//Communication error
	fbKommTof(IN:=bError , PT:=T#20S , Q=> , ET=> );
	fbKommTon(bInput:=fbKommTof.Q , tAlarmDelay:=T#1M , bAutoReset:= , bAlarmOutput=> );
	FAULT :=fbKommTon.bAlarmOutput;
		
//Write busy	
	oaksgvl.aBModbusBusyFlagga[modbusTCP.iModbusLoop,nUnitID] := bBusy;

METHOD mAnalogToRaw : WORD
VAR_INPUT
	rValueToConvert : REAL; //Rå-värde
END_VAR

VAR
	x1 : REAL;
	x2 : REAL;
	y1 : REAL;
	y2 : REAL;
	rPercent : REAL;
	rRawAnalog : REAL;
	rInternalVal: REAL;
END_VAR
//0-100%
rInternalVal := LIMIT(0,rValueToConvert,100);

x1 := 0; 
x2 := 100; 
y1 := 0; 
y2 := 10;
rPercent := fScale2p(rInternalVal,y1, y2, x1, x2);

//0-10V
x1 := 0; 
x2 := 10.24; 
y1 := 0; 
y2 := 32767;
rRawAnalog := fScale2p(rPercent, y1, y2, x1, x2);
mAnalogToRaw := fRealtoWord(rRawAnalog, 1);
END_METHOD

METHOD mAnalogToRawFallback : WORD
VAR_INPUT
	rValueToConvert : REAL; //Rå-värde
END_VAR

VAR
	x1 : REAL;
	x2 : REAL;
	y1 : REAL;
	y2 : REAL;
	rPercent : REAL;
	rRawAnalog : REAL;
	rInternalVal: REAL;
END_VAR
//0-100%
rInternalVal := LIMIT(0,rValueToConvert,100);

//0-10V
x1 := 0; 
x2 := 10.24; 
y1 := 0; 
y2 := 32767;

mAnalogToRawFallback := fRealtoWord(fScale2p(rInternalVal, y1, y2, x1, x2), 1);
END_METHOD

METHOD mRawToAnalog : REAL
VAR_INPUT
	rValueToConvert : WORD; //Rå-värde
END_VAR

VAR
	x1 : REAL;
	x2 : REAL;
	y1 : REAL;
	y2 : REAL;
	rTemp : REAL;
END_VAR
//0-10V
rTemp := fSignedConverter(rValueToConvert);

x1 := 0; 
x2 := 32767;
y1 := 0; 
y2 := 10.24; 
mRawToAnalog := fScale2p(rTemp, y1, y2, x1, x2);
END_METHOD

END_FUNCTION_BLOCK

// oaksModbusLibrary/Metz/fbMetzMR_MULTI
//Oaks AB
//2023-09-19 / Johan Bornemyr
//Funktionsblock för hantering av Metz MR IO-system. 
//MR-MULTI. Modul med 29 IO. Fysisk handställningsmöjlighet 0-10V på modul.
FUNCTION_BLOCK fbMetzMR_MULTI
VAR_INPUT
	bEnable : BOOL := TRUE; //Aktivering
	modbusTCP : ST_ModbusTCP;
	nUnitID: BYTE := 0;
	
	bDO1 : BOOL := FALSE; //Manöver digital utgång 1
	bDO1fallback : BOOL; //Värde vid komm.fel utgång 1
	bDO2 : BOOL := FALSE; //Manöver digital utgång 2
	bDO2fallback : BOOL; //Värde vid komm.fel utgång 2
	bDO3 : BOOL := FALSE; //Manöver digital utgång 3
	bDO3fallback : BOOL; //Värde vid komm.fel utgång 3
	bDO4 : BOOL := FALSE; //Manöver digital utgång 4
	bDO4fallback : BOOL; //Värde vid komm.fel utgång 4
	bTransistorDO1 : BOOL := FALSE; //Manöver digital Transistorutgång 1
	bTransistorDO1fallback : BOOL; //Värde vid komm.fel Transistorutgång 1
	bTransistorDO2 : BOOL := FALSE; //Manöver digital Transistorutgång 2
	bTransistorDO2fallback : BOOL; //Värde vid komm.fel Transistorutgång 2
	bTransistorDO3 : BOOL := FALSE; //Manöver digital Transistorutgång 3
	bTransistorDO3fallback : BOOL; //Värde vid komm.fel Transistorutgång 3
	bTransistorDO4 : BOOL := FALSE; //Manöver digital Transistorutgång 4
	bTransistorDO4fallback : BOOL; //Värde vid komm.fel Transistorutgång 4
	rAO1Setpoint : REAL := 0; //Börvärde Analog utgång 1 (0-100%)
	rAO1FallbackVoltage : REAL := 0; //Börvärde Analog utgång 1 (0-10V)
	rAO2Setpoint : REAL := 0; //Börvärde Analog utgång 2 (0-100%)
	rAO2FallbackVoltage : REAL := 0; //Börvärde Analog utgång 2 (0-10V)
	sensor1config : ST_MetzAI8config;
	sensor2config : ST_MetzAI8config;
	sensor3config : ST_MetzAI8config;
	sensor4config : ST_MetzAI8config;
	sensor5config : ST_MetzAI8config;
	sensor6config : ST_MetzAI8config;
END_VAR
	
VAR_INPUT PERSISTENT
	SP1 AT %M* : REAL := 0;//Komm.fels fördröjning IO~wp:[unit]ms[format]0.0
END_VAR

VAR_OUTPUT
	DI1_V AT %M* : BOOL;//Digital ingång 1~wp:
	DI2_V AT %M* : BOOL;//Digital ingång 2~wp:
	DI3_V AT %M* : BOOL;//Digital ingång 3~wp:
	DI4_V AT %M* : BOOL;//Digital ingång 4~wp:
	DI5_V AT %M* : BOOL;//Digital ingång 5~wp:
	DI6_V AT %M* : BOOL;//Digital ingång 6~wp:
	DI7_V AT %M* : BOOL;//Digital ingång 7~wp:
	DI8_V AT %M* : BOOL;//Digital ingång 8~wp:
	DI9_V AT %M* : BOOL;//Digital ingång 9~wp:
	DI10_V AT %M* : BOOL;//Digital ingång 10~wp:
	DI11_V AT %M* : BOOL;//Digital ingång 11~wp:
	DI12_V AT %M* : BOOL;//Digital ingång 12~wp:
	
	DO1_V AT %M* : BOOL :=FALSE;//Digital utgång 1~wp:
	DO2_V AT %M* : BOOL :=FALSE;//Digital utgång 2~wp:
	DO3_V AT %M* : BOOL :=FALSE;//Digital utgång 3~wp:
	DO4_V AT %M* : BOOL :=FALSE;//Digital utgång 4~wp:
	
	TRANSISTOR_DO1_V AT %M* : BOOL :=FALSE;//Digital utgång 1~wp:
	TRANSISTOR_DO2_V AT %M* : BOOL :=FALSE;//Digital utgång 2~wp:
	TRANSISTOR_DO3_V AT %M* : BOOL :=FALSE;//Digital utgång 3~wp:
	TRANSISTOR_DO4_V AT %M* : BOOL :=FALSE;//Digital utgång 4~wp:
	
	
	AI1_PV AT %M* : REAL; //Råvärde utgång 1~wp:[format]0.00
	AI1_PV1 AT %M* : STRING;//Konfigurering ingång 1~wp:
	sensor1 : ST_MetzAI8Sensor; //Skicka till sensorblock
	AI2_PV AT %M* : REAL; //Råvärde utgång 2~wp:[format]0.00
	AI2_PV1 AT %M* : STRING;//Konfigurering ingång 2~wp:
	sensor2 : ST_MetzAI8Sensor; //Skicka till sensorblock
	AI3_PV AT %M* : REAL; //Råvärde utgång 3~wp:[format]0.00
	AI3_PV1 AT %M* : STRING;//Konfigurering ingång 3~wp:
	sensor3 : ST_MetzAI8Sensor; //Skicka till sensorblock
	AI4_PV AT %M* : REAL; //Råvärde utgång 4~wp:[format]0.00
	AI4_PV1 AT %M* : STRING;//Konfigurering ingång 4~wp:
	sensor4 : ST_MetzAI8Sensor; //Skicka till sensorblock
	AI5_PV AT %M* : REAL; //Råvärde utgång 5~wp:[format]0.00
	AI5_PV1 AT %M* : STRING;//Konfigurering ingång 5~wp:
	sensor5 : ST_MetzAI8Sensor; //Skicka till sensorblock
	AI6_PV AT %M* : REAL; //Råvärde utgång 6~wp:[format]0.00
	AI6_PV1 AT %M* : STRING;//Konfigurering ingång 6~wp:
	sensor6 : ST_MetzAI8Sensor; //Skicka till sensorblock
	
	AO1_OP AT %M* : REAL;//Analog utgång 1~wp:[unit]V[format]0.00
	AO1_FAULT AT %M* : BOOL;//Omkopplare i fel läge utgång 1~wp:
	AO2_OP AT %M* : REAL;//Analog utgång 2~wp:[unit]V[format]0.00
	AO2_FAULT AT %M* : BOOL;//Omkopplare i fel läge utgång 2~wp:
	
	PV8 AT %M* : STRING;//Modbus konfiguering~wp:
	FAULT AT %M* : BOOL;//Kommunikationsfel~wp:
END_VAR
VAR
	//Communication error
	fbKommTof : tof; 
	fbKommTon : fbAlarm;	

	tTimeOut : TIME :=T#5S;
	sIP: STRING(255);
	sPort: STRING(255);
	sModbusID: STRING(255);
	sModbusLoop: STRING(255);
	sTemp : STRING(255);	

	bSekvensFlagga : BOOL;
	R_TRIG_Sekvens: R_TRIG;
(*************** DIGITAL IN - START ***************)	
	FB_MBReadRegs_InputRegsDigitalIn: FB_MBReadInputRegs;
	wInputRegsDigitalIn : WORD; //Read input regs modbus function 4. 	
(*************** DIGITAL IN - SLUT ***************)
(*************** DIGITAL UT - START ***************)
	iStep: INT;
	bError: BOOL;
	bBusy: BOOL;
	
	//Read output values and default values
	FB_MBReadRegs_ArrHolding1: FB_MBReadRegs;
	ArrHolding1 : ARRAY [0..7] OF WORD; //Holding


	fbReadWriteHoldingRegReal_ComError: fbReadWriteHoldingRegReal;
	
	//Configuration
	FB_MBWriteRegs_Config: FB_MBWriteSingleReg;
	wWriteConfig : WORD; //Läs/skriv input regs modbus function 4.
	wReadConfig : WORD; //Läs/skriv input regs modbus function 4.
		
	//Outputs
	FB_MBWriteRegs_Outputs: FB_MBWriteSingleReg;
	wWriteOutputs : WORD; //Läs/skriv input regs modbus function 6.
(*************** DIGITAL UT - SLUT ***************)
(*************** ANALOG UT - START ***************)
	iStepAnalogOut: INT;
	bErrorAnalogOutput: BOOL;
	bBusyAnalogOutput: BOOL;
	
	//Read output values and default values
	FB_MBReadRegs_ArrHoldingAnalogOutput: FB_MBReadRegs;
	ArrHoldingAnalogOutput : ARRAY [0..3] OF WORD; //Holding

	//Outputs in manual mode
	FB_MBReadInputs_wDiscreteInputsAnalogOutput: FB_MBReadInputs;
	wDiscreteInputsAnalogOutput : WORD; //Discrete Input;
	
	fbAlarm_Output1manAnalogOutput : fbAlarm;
	fbAlarm_Output2manAnalogOutput : fbAlarm;

	fbReadWriteHoldingRegReal_ComErrorAnalogOutput: fbReadWriteHoldingRegReal;
	
	//Configuration
	FB_MBWriteRegs_ConfigAnalogOutput: FB_MBWriteRegs;
	wInputRegs2wAnalogOutput : ARRAY[1..2] OF WORD; //Läs/skriv input regs modbus function 16.
	wInputRegs2rAnalogOutput : ARRAY[1..2] OF WORD; //Läs/skriv input regs modbus function 16.
	iConfigChangedAnalogOutput: INT;
	bChangeConfigAnalogOutput: BOOL;
	arrIndexAnalogOutput: INT;
	
	//Outputs
	FB_MBWriteRegs_AnalogOutput: FB_MBWriteRegs;
	wInputRegsOutputswAnalogOutput : ARRAY[1..2] OF WORD; //Läs/skriv input regs modbus function 16.
(*************** ANALOG UT - SLUT ***************)	
(*************** ANALOG IN - START ***************)		
	iStepAnalogIn: INT;
	bErrorAnalogIn: BOOL;
	bBusyAnalogIn: BOOL;	

	//Configuration
	FB_MBReadInputRegs_ValuesAnalogIn: FB_MBReadInputRegs;
	wInputRegsValuesAnalogIn : ARRAY[0..11] OF WORD; //Läs input regs modbus function 4.
	wHoldingRegs2writeConfigAnalogIn : ARRAY[16..21] OF WORD; //Läs/skriv input regs modbus function 16.
	wHoldingRegs2readConfigAnalogIn : ARRAY[16..21] OF WORD; //Läs/skriv input regs modbus function 16.
	
	FB_MBWriteRegs_ConfigAnalogIn: FB_MBWriteRegs;
	FB_MBReadRegs_ConfigAnalogIn: FB_MBReadRegs;
	arrIndexAnalogIn: INT;
	iConfigChangedAnalogIn: INT;
	bChangeConfigAnalogIn: BOOL;

	//Convert to float
	wTempArrayConvertingFromFloatAnalogIn: ARRAY[0..1] OF WORD; // Används för att byta ordning på de två 16-bitars registerna som float-värdet består utav.
(*************** ANALOG IN - SLUT ***************)	
END_VAR

//Sekvens	
	R_TRIG_Sekvens(CLK:= oaksGVL.aBModbusSekvens[modbusTCP.iModbusLoop] = BYTE_TO_INT(nUnitID), Q=> bSekvensFlagga);
	
	
//Modbus config
	sIP := CONCAT (modbusTCP.sIPAddr, '');
	sPort := CONCAT ('<br>Port: ', UINT_TO_STRING(modbusTCP.nTCPPort)); 								
	sModbusID := CONCAT('<br>ID: ', BYTE_TO_STRING(nUnitID));
	sModbusLoop := CONCAT('<br>Loop: ', INT_TO_STRING(modbusTCP.iModbusLoop));	

	sTemp := sIP;
	sTemp := CONCAT(sTemp, sPort);
	sTemp := CONCAT(sTemp, sModbusID);
	sTemp := CONCAT(sTemp, sModbusLoop);
	
	PV8 := sTemp;
	
	mDigitalIn();
	mDigitalOut();
	mAnalogIn();
	mAnalogOut();
	

//Communication error
	fbKommTof(IN:=bErrorAnalogOutput , PT:=T#20S , Q=> , ET=> );
	fbKommTon(bInput:=fbKommTof.Q , tAlarmDelay:=T#1M , bAutoReset:= , bAlarmOutput=> );
	FAULT :=fbKommTon.bAlarmOutput;
		
//Write busy	
	oaksgvl.aBModbusBusyFlagga[modbusTCP.iModbusLoop,nUnitID] := bBusyAnalogOutput;

METHOD PRIVATE config : WORD
VAR_INPUT
	bResistance : BOOL; //0-10V (false) eller resistans (true)
	wSensorType : WORD;
	
END_VAR

VAR
	wOffset : WORD := 0; 
END_VAR
//Temperaturmätning
IF bResistance THEN

	wOffset := wSensorType;
	
	config.0 := FALSE; //Float
	config.1 := wOffset.0; 
	config.2 := wOffset.1; 
	config.3 := wOffset.2; 
	config.4 := wOffset.3;  
	config.5 := wOffset.4; 
	config.6 := wOffset.5; 
	config.7 := TRUE; //Välj resistans 
	config.8 := FALSE; 
	config.9 := FALSE; 
	config.10 := FALSE; 
	config.11 := FALSE; 
	config.12 := FALSE; 
	config.13 := FALSE; 
	config.14 := FALSE; 
	config.15 := FALSE; 
 
  
//Spänningsmätning
ELSE
	config.0 := FALSE; //Float
	config.1 := FALSE; 
	config.2 := FALSE; 
	config.3 := FALSE; 
	config.4 := FALSE;  
	config.5 := FALSE; 
	config.6 := FALSE; 
	config.7 := FALSE; //Välj resistans 
	config.8 := FALSE; 
	config.9 := FALSE; 
	config.10 := FALSE; 
	config.11 := FALSE; 
	config.12 := FALSE; 
	config.13 := FALSE; 
	config.14 := FALSE; 
	config.15 := FALSE; 
END_IF
END_METHOD

METHOD PRIVATE mAnalogIn
VAR_INPUT
END_VAR
	CASE iStepAnalogIn OF

	0: 	//Start/reset
		bBusyAnalogIn := FALSE;
				
		IF bEnable AND bSekvensFlagga THEN
			iStepAnalogIn := 1;
			bErrorAnalogIn := FALSE;
		END_IF
		
	1: 	//Read measured values
		bBusyAnalogIn := TRUE;
			
		FB_MBReadInputRegs_ValuesAnalogIn.bExecute := TRUE;
	
		FB_MBReadInputRegs_ValuesAnalogIn(
		sIPAddr:= modbusTCP.sIpAddr, 
		nTCPPort:= modbusTCP.nTCPPort, 
		nUnitID:= nUnitID, 
		nQuantity:= 12,
		nMBAddr:= 0, 
		cbLength:= SIZEOF(wInputRegsValuesAnalogIn), 
		pDestAddr:= ADR(wInputRegsValuesAnalogIn), 
		bExecute:= , 
		tTimeout:= tTimeOut, 
		bBusy=> , 
		bError=> , 
		nErrId=> , 
		cbRead=> );
		
		//Ingång 1
		wTempArrayConvertingFromFloatAnalogIn[0] := wInputRegsValuesAnalogIn[1];
		wTempArrayConvertingFromFloatAnalogIn[1] := wInputRegsValuesAnalogIn[0]; 

		
		AI1_PV := fWordToReal(wTempArrayConvertingFromFloatAnalogIn);
		
		IF sensor1config.bResistance THEN
			AI1_PV := fWordToReal(wTempArrayConvertingFromFloatAnalogIn);
			AI1_PV1 := CONCAT('Givartyp: ', TO_STRING(sensor1config.sensorType));
		ELSE
			stemp := '0-10V';
			AI1_PV1 := sTemp;
		END_IF
		
		//Info till sensorblock
		sensor1.bComError := FAULT;
		sensor1.rRawValue := AI1_PV;
		sensor1.sSensorConfig := AI1_PV1;
		
		//Ingång 2
		wTempArrayConvertingFromFloatAnalogIn[0] := wInputRegsValuesAnalogIn[3];
		wTempArrayConvertingFromFloatAnalogIn[1] := wInputRegsValuesAnalogIn[2];
		
		AI2_PV := fWordToReal(wTempArrayConvertingFromFloatAnalogIn);
		
		IF sensor2config.bResistance THEN
			AI2_PV1 := CONCAT('Givartyp: ', TO_STRING(sensor2config.sensorType));
		ELSE
			stemp := '0-10V';
			AI2_PV1 := sTemp; 
  
		END_IF
		
		//Info till sensorblock
		sensor2.bComError := FAULT;
		sensor2.rRawValue := AI2_PV;
		sensor2.sSensorConfig := AI2_PV1;
		
		//Ingång 3
		wTempArrayConvertingFromFloatAnalogIn[0] := wInputRegsValuesAnalogIn[5];
		wTempArrayConvertingFromFloatAnalogIn[1] := wInputRegsValuesAnalogIn[4];
		
		AI3_PV := fWordToReal(wTempArrayConvertingFromFloatAnalogIn);
		
		IF sensor3config.bResistance THEN
			AI3_PV1 := CONCAT('Givartyp: ', TO_STRING(sensor3config.sensorType));
		ELSE
			stemp := '0-10V';
			AI3_PV1 := sTemp; 
		END_IF
		
		//Info till sensorblock
		sensor3.bComError := FAULT;
		sensor3.rRawValue := AI3_PV;
		sensor3.sSensorConfig := AI3_PV1;
		
		//Ingång 4
		wTempArrayConvertingFromFloatAnalogIn[0] := wInputRegsValuesAnalogIn[7];
		wTempArrayConvertingFromFloatAnalogIn[1] := wInputRegsValuesAnalogIn[6];
		
		AI4_PV := fWordToReal(wTempArrayConvertingFromFloatAnalogIn);
		
		IF sensor4config.bResistance THEN
			AI4_PV1 := CONCAT('Givartyp: ', TO_STRING(sensor4config.sensorType));
		ELSE
			stemp := '0-10V';
			AI4_PV1 := sTemp;
		END_IF
		
		//Info till sensorblock
		sensor4.bComError := FAULT;
		sensor4.rRawValue := AI4_PV;
		sensor4.sSensorConfig := AI4_PV1;
		
		//Ingång 5
		wTempArrayConvertingFromFloatAnalogIn[0] := wInputRegsValuesAnalogIn[9];
		wTempArrayConvertingFromFloatAnalogIn[1] := wInputRegsValuesAnalogIn[8];

		AI5_PV := fWordToReal(wTempArrayConvertingFromFloatAnalogIn);
	
		IF sensor5config.bResistance THEN
			AI5_PV1 := CONCAT('Givartyp: ', TO_STRING(sensor5config.sensorType));
		ELSE
			stemp := '0-10V';
			AI5_PV1 := sTemp;
		END_IF
		
		//Info till sensorblock
		sensor5.bComError := FAULT;
		sensor5.rRawValue := AI5_PV;
		sensor5.sSensorConfig := AI5_PV1;
		
		//Ingång 6
		wTempArrayConvertingFromFloatAnalogIn[0] := wInputRegsValuesAnalogIn[11];
		wTempArrayConvertingFromFloatAnalogIn[1] := wInputRegsValuesAnalogIn[10]; 
		
		AI6_PV := fWordToReal(wTempArrayConvertingFromFloatAnalogIn);
				
		IF sensor6config.bResistance THEN
			AI6_PV1 := CONCAT('Givartyp: ', TO_STRING(sensor6config.sensorType));
		ELSE
			stemp := '0-10V';
			AI6_PV1 := sTemp;
		END_IF
		
		//Info till sensorblock
		sensor6.bComError := FAULT;
		sensor6.rRawValue := AI6_PV;
		sensor6.sSensorConfig := AI6_PV1;
		
		//Error 
		IF FB_MBReadInputRegs_ValuesAnalogIn.bError THEN
			FB_MBReadInputRegs_ValuesAnalogIn(bExecute := FALSE);
			iStepAnalogIn := 99;
		END_IF
	
		//Gå till nästa steg
		IF NOT FB_MBReadInputRegs_ValuesAnalogIn.bBusy AND NOT FB_MBReadInputRegs_ValuesAnalogIn.bError THEN
			FB_MBReadInputRegs_ValuesAnalogIn(bExecute := FALSE);
			bErrorAnalogIn := FALSE;
			iStepAnalogIn := 2;
		END_IF;
		
	2: 	//Läs config
		bBusyAnalogIn := TRUE;
		FB_MBReadRegs_ConfigAnalogIn.bExecute := TRUE;
	
		//Konfigurering
		wHoldingRegs2writeConfigAnalogIn[16] := config(sensor1config.bResistance,sensor1config.sensorType);
		wHoldingRegs2writeConfigAnalogIn[17] := config(sensor2config.bResistance,sensor2config.sensorType);
		wHoldingRegs2writeConfigAnalogIn[18] := config(sensor3config.bResistance,sensor3config.sensorType);
		wHoldingRegs2writeConfigAnalogIn[19] := config(sensor4config.bResistance,sensor4config.sensorType);
		wHoldingRegs2writeConfigAnalogIn[20] := config(sensor5config.bResistance,sensor5config.sensorType);
		wHoldingRegs2writeConfigAnalogIn[21] := config(sensor6config.bResistance,sensor6config.sensorType);
	
		FB_MBReadRegs_ConfigAnalogIn(
		sIPAddr:= modbusTCP.sIpAddr, 
		nTCPPort:= modbusTCP.nTCPPort, 
		nUnitID:= nUnitID, 
		nQuantity:= 6, 
		nMBAddr:= 16, 
		cbLength:= SIZEOF(wHoldingRegs2readConfigAnalogIn), 
		pDestAddr:= ADR(wHoldingRegs2readConfigAnalogIn), 
		bExecute:= , 
		tTimeout:= tTimeOut, 
		bBusy=> , 
		bError=> , 
		nErrId=> , 
		cbRead=> );

		//Error 
		IF FB_MBReadRegs_ConfigAnalogIn.bError THEN
			FB_MBReadRegs_ConfigAnalogIn(bExecute := FALSE);
			iStepAnalogIn := 99;
		END_IF
	
		//Next step
		IF NOT FB_MBReadRegs_ConfigAnalogIn.bBusy AND NOT FB_MBReadRegs_ConfigAnalogIn.bError THEN
			FB_MBReadRegs_ConfigAnalogIn(bExecute := FALSE);
		
			//Loop to check if config is different
			FOR arrIndexAnalogIn:=16 TO 21 BY 1 DO
				IF wHoldingRegs2readConfigAnalogIn[arrIndexAnalogIn] = wHoldingRegs2writeConfigAnalogIn[arrIndexAnalogIn] THEN
			 		iConfigChangedAnalogIn := iConfigChangedAnalogIn;
				ELSE 
			 		iConfigChangedAnalogIn := iConfigChangedAnalogIn +1;
				END_IF
			END_FOR;
	
			IF iConfigChangedAnalogIn > 0 THEN
				bChangeConfigAnalogIn := TRUE;
				iStepAnalogIn := 3;
				bErrorAnalogIn := FALSE;
			ELSE 
				iStepAnalogIn := 4;
				bErrorAnalogIn := FALSE;
			END_IF
				
		END_IF;
	
	3: //Write if config is different from read value
		bBusyAnalogIn := TRUE;	
		IF bChangeConfigAnalogIn THEN
			FB_MBWriteRegs_ConfigAnalogIn.bExecute := TRUE;
		END_IF
			
		FB_MBWriteRegs_ConfigAnalogIn(
		sIPAddr:= modbusTCP.sIpAddr, 
		nTCPPort:= modbusTCP.nTCPPort, 
		nUnitID:= nUnitID, 
		nQuantity:= 6, 
		nMBAddr:= 16, 
		cbLength:= SIZEOF(wHoldingRegs2writeConfigAnalogIn), 
		pSrcAddr:= ADR(wHoldingRegs2writeConfigAnalogIn), 
		bExecute:=, 
		tTimeout:= tTimeOut, 
		bBusy=> , 
		bError=> , 
		nErrId=> );
		
		IF FB_MBWriteRegs_ConfigAnalogIn.bError THEN
			FB_MBWriteRegs_ConfigAnalogIn(bExecute := FALSE);
			iStepAnalogIn := 99;
		END_IF
	
		//Next step
		IF NOT FB_MBWriteRegs_ConfigAnalogIn.bBusy AND NOT FB_MBWriteRegs_ConfigAnalogIn.bError THEN
			FB_MBWriteRegs_ConfigAnalogIn(bExecute := FALSE);
			iConfigChangedAnalogIn := 0;
			bChangeConfigAnalogIn := FALSE; //Reset write
			bErrorAnalogIn := FALSE;
			iStepAnalogIn := 4;
		END_IF;
			
	4: //Done
		bBusyAnalogIn := FALSE;
		iStepAnalogIn := 0;

	99: //Error handling
		bBusyAnalogIn := FALSE;
		bErrorAnalogIn := TRUE;
		iStepAnalogIn := 0;
		
END_CASE
END_METHOD

METHOD PRIVATE mAnalogOut
VAR_INPUT
END_VAR
	CASE iStepAnalogOut OF

	0: 	//Start/reset
		bBusyAnalogOutput := FALSE;

		IF bEnable AND bSekvensFlagga THEN
			iStepAnalogOut := 1;
			bErrorAnalogOutput := FALSE;
		END_IF
		
	1: 	//Read measured values
		bBusyAnalogOutput := TRUE;
		
		FB_MBReadInputs_wDiscreteInputsAnalogOutput.bExecute := TRUE;

		FB_MBReadInputs_wDiscreteInputsAnalogOutput(
		sIPAddr:= modbusTCP.sIpAddr, 
		nTCPPort:= modbusTCP.nTCPPort, 
		nUnitID:= nUnitID, 
		nQuantity:= 4, 
		nMBAddr:= 0, 
		cbLength:= SIZEOF(wDiscreteInputsAnalogOutput), 
		pDestAddr:= ADR(wDiscreteInputsAnalogOutput),
		bExecute:=, 
		tTimeout:= tTimeOut, 
		bBusy=> , 
		bError=> , 
		nErrId=> , 
		cbRead=> );
	
		//Switch manual alarm
		fbAlarm_Output1manAnalogOutput(bInput:= wDiscreteInputsAnalogOutput.0, tAlarmDelay:= T#3S, bAutoReset:= , bAlarmOutput=> AO1_FAULT);
		fbAlarm_Output2manAnalogOutput(bInput:= wDiscreteInputsAnalogOutput.1, tAlarmDelay:= T#3S, bAutoReset:= , bAlarmOutput=> AO2_FAULT);
			
		//Error 
		IF FB_MBReadInputs_wDiscreteInputsAnalogOutput.bError THEN
			FB_MBReadInputs_wDiscreteInputsAnalogOutput(bExecute := FALSE);
			iStepAnalogOut := 99;
		END_IF
	
		//Next step
		IF NOT FB_MBReadInputs_wDiscreteInputsAnalogOutput.bBusy AND NOT FB_MBReadInputs_wDiscreteInputsAnalogOutput.bError THEN
			FB_MBReadInputs_wDiscreteInputsAnalogOutput(bExecute := FALSE);
			bErrorAnalogOutput := FALSE;
			iStepAnalogOut := 2;
		END_IF;
			
		
	2: //Read Data (Value on output)
		bBusyAnalogOutput := TRUE;
		FB_MBReadRegs_ArrHoldingAnalogOutput.bExecute := TRUE;

		//Read Holding 0-7
		FB_MBReadRegs_ArrHoldingAnalogOutput(
		sIPAddr:= modbusTCP.sIpAddr, 
		nTCPPort:= modbusTCP.nTCPPort, 
		nUnitID:= nUnitID, 
		nQuantity:= 4, 
		nMBAddr:= 74, 
		cbLength:= SIZEOF(ArrHoldingAnalogOutput), 
		pDestAddr:= ADR(ArrHoldingAnalogOutput), 
		bExecute:=, 
		tTimeout:= tTimeOut, 
		bBusy=> ,
		bError=> , 
		nErrId=> , 
		cbRead=> );
	
		//Values
		AO1_OP := mRawToAnalog(ArrHoldingAnalogOutput[0]); //0
		AO2_OP := mRawToAnalog(ArrHoldingAnalogOutput[1]); //1

		//Error 
		IF FB_MBReadRegs_ArrHoldingAnalogOutput.bError THEN
			FB_MBReadRegs_ArrHoldingAnalogOutput(bExecute := FALSE);
			iStepAnalogOut := 99;
		END_IF
	
		//Gå till nästa steg
		IF NOT FB_MBReadRegs_ArrHoldingAnalogOutput.bBusy AND NOT FB_MBReadRegs_ArrHoldingAnalogOutput.bError THEN
			FB_MBReadRegs_ArrHoldingAnalogOutput(bExecute := FALSE);
			bErrorAnalogOutput := FALSE;
			iStepAnalogOut := 3;
		END_IF;

	3: //Read/Write communication error timedelay (config)
		bBusyAnalogOutput := TRUE;

		//User input
		IF SP1 < 0 THEN
			SP1 := 0;
		END_IF;
		
		IF SP1 > 65535 THEN
			SP1 := 655;
		END_IF;
		
		fbReadWriteHoldingRegReal_ComErrorAnalogOutput.bEnable := TRUE;
		
		fbReadWriteHoldingRegReal_ComErrorAnalogOutput(
		sIPAddr:= modbusTCP.sIpAddr, 
		nTCPPort:= modbusTCP.nTCPPort, 
		nUnitID:= nUnitID, 
		mBusAdr:= 66, 
		bEnable:= , 
		tTimeout:= tTimeOut, 
		rReal:= SP1, 
		uiFaktor:= 100, 
		bError=> , 
		bBusy=> , 
		bSuccess=> );
				
		//Error 
		IF fbReadWriteHoldingRegReal_ComErrorAnalogOutput.bError THEN
			fbReadWriteHoldingRegReal_ComErrorAnalogOutput(bEnable := FALSE);
			iStepAnalogOut := 99;
		END_IF
	
		//Gå till nästa steg
		IF NOT fbReadWriteHoldingRegReal_ComErrorAnalogOutput.bBusy AND NOT fbReadWriteHoldingRegReal_ComErrorAnalogOutput.bError THEN
			fbReadWriteHoldingRegReal_ComErrorAnalogOutput(bEnable := FALSE);
			bErrorAnalogOutput := FALSE;
			iStepAnalogOut := 4;
		END_IF;

	4:	//Read/Write default values (config)
		
		//Config in IO
		wInputRegs2rAnalogOutput[1] := ArrHoldingAnalogOutput[2]; //3;
		wInputRegs2rAnalogOutput[2] := ArrHoldingAnalogOutput[3]; //4;
		//Config in PLC	
		wInputRegs2wAnalogOutput[1] := mAnalogToRawFallback(rAO1FallbackVoltage); //3;
		wInputRegs2wAnalogOutput[2] := mAnalogToRawFallback(rAO2FallbackVoltage); //4;
		
		FOR arrIndexAnalogOutput:=1 TO 2 BY 1 DO
				IF wInputRegs2rAnalogOutput[arrIndexAnalogOutput] = wInputRegs2wAnalogOutput[arrIndexAnalogOutput] THEN
			 		iConfigChangedAnalogOutput := iConfigChangedAnalogOutput;
				ELSE 
			 		iConfigChangedAnalogOutput := iConfigChangedAnalogOutput +1;
				END_IF
		END_FOR;
	
		IF iConfigChangedAnalogOutput > 0 THEN
			bChangeConfigAnalogOutput := TRUE;
			iStepAnalogOut := 5;
			bErrorAnalogOutput := FALSE;
		ELSE 
			iStepAnalogOut := 6;
			bErrorAnalogOutput := FALSE;
		END_IF
 
	5: //Write if config is different from read value
		bBusyAnalogOutput := TRUE;	
		IF bChangeConfigAnalogOutput THEN
			FB_MBWriteRegs_ConfigAnalogOutput.bExecute := TRUE;
		END_IF
			
		FB_MBWriteRegs_ConfigAnalogOutput(
		sIPAddr:= modbusTCP.sIpAddr, 
		nTCPPort:= modbusTCP.nTCPPort, 
		nUnitID:= nUnitID, 
		nQuantity:= 2, 
		nMBAddr:= 78, 
		cbLength:= SIZEOF(wInputRegs2wAnalogOutput), 
		pSrcAddr:= ADR(wInputRegs2wAnalogOutput), 
		bExecute:=, 
		tTimeout:= tTimeOut, 
		bBusy=> , 
		bError=> , 
		nErrId=> );
		
		IF FB_MBWriteRegs_ConfigAnalogOutput.bError THEN
			FB_MBWriteRegs_ConfigAnalogOutput(bExecute := FALSE);
			iStepAnalogOut := 99;
		END_IF
	
		//Next step
		IF NOT FB_MBWriteRegs_ConfigAnalogOutput.bBusy AND NOT FB_MBWriteRegs_ConfigAnalogOutput.bError THEN
			FB_MBWriteRegs_ConfigAnalogOutput(bExecute := FALSE);
			iConfigChangedAnalogOutput := 0;
			bChangeConfigAnalogOutput := FALSE; //Reset write
			bErrorAnalogOutput := FALSE;
			iStepAnalogOut := 6;
		END_IF;

	6: //Write outputs
		bBusyAnalogOutput := TRUE;	
			
		wInputRegsOutputswAnalogOutput[1] := mAnalogToRaw(rAO1Setpoint);
		wInputRegsOutputswAnalogOutput[2] := mAnalogToRaw(rAO2Setpoint);
		
		FB_MBWriteRegs_AnalogOutput.bExecute := TRUE;
		
		FB_MBWriteRegs_AnalogOutput(
		sIPAddr:= modbusTCP.sIpAddr, 
		nTCPPort:= modbusTCP.nTCPPort, 
		nUnitID:= nUnitID, 
		nQuantity:= 2, 
		nMBAddr:= 74, 
		cbLength:= SIZEOF(wInputRegsOutputswAnalogOutput), 
		pSrcAddr:= ADR(wInputRegsOutputswAnalogOutput), 
		bExecute:=, 
		tTimeout:= tTimeOut, 
		bBusy=> , 
		bError=> , 
		nErrId=> );
		
		IF FB_MBWriteRegs_AnalogOutput.bError THEN
			FB_MBWriteRegs_AnalogOutput(bExecute := FALSE);
			iStepAnalogOut := 99;
		END_IF
	
		//Next step
		IF NOT FB_MBWriteRegs_AnalogOutput.bBusy AND NOT FB_MBWriteRegs_AnalogOutput.bError THEN
			FB_MBWriteRegs_AnalogOutput(bExecute := FALSE);
			bErrorAnalogOutput := FALSE;
			iStepAnalogOut := 20;
		END_IF;

	20: //Done
		bBusyAnalogOutput := FALSE;
		iStepAnalogOut := 0;

	99: //Error handling
		bBusyAnalogOutput := FALSE;
		bErrorAnalogOutput := TRUE;
		iStepAnalogOut := 0;
		
END_CASE
END_METHOD

METHOD mAnalogToRaw : WORD
VAR_INPUT
	rValueToConvert : REAL; //Rå-värde
END_VAR

VAR
	x1 : REAL;
	x2 : REAL;
	y1 : REAL;
	y2 : REAL;
	rPercent : REAL;
	rRawAnalog : REAL;
	rInternalVal: REAL;
END_VAR
//0-100%
rInternalVal := LIMIT(0,rValueToConvert,100);

x1 := 0; 
x2 := 100; 
y1 := 0; 
y2 := 10;
rPercent := fScale2p(rInternalVal,y1, y2, x1, x2);

//0-10V
x1 := 0; 
x2 := 10.24; 
y1 := 0; 
y2 := 32767;
rRawAnalog := fScale2p(rPercent, y1, y2, x1, x2);
mAnalogToRaw := fRealtoWord(rRawAnalog, 1);
END_METHOD

METHOD mAnalogToRawFallback : WORD
VAR_INPUT
	rValueToConvert : REAL; //Rå-värde
END_VAR

VAR
	x1 : REAL;
	x2 : REAL;
	y1 : REAL;
	y2 : REAL;
	rPercent : REAL;
	rRawAnalog : REAL;
	rInternalVal: REAL;
END_VAR
//0-100%
rInternalVal := LIMIT(0,rValueToConvert,100);

x1 := 0; 
x2 := 100; 
y1 := 0; 
y2 := 10;
rPercent := fScale2p(rInternalVal,y1, y2, x1, x2);

//0-10V
x1 := 0; 
x2 := 10.24; 
y1 := 0; 
y2 := 32767;

mAnalogToRawFallback := fRealtoWord(fScale2p(rPercent, y1, y2, x1, x2), 1);
END_METHOD

METHOD PRIVATE mDigitalIn
VAR_INPUT
END_VAR
	//Read Input states
	FB_MBReadRegs_InputRegsDigitalIn(
	sIPAddr:= modbusTCP.sIpAddr, 
	nTCPPort:= modbusTCP.nTCPPort, 
	nUnitID:= nUnitID, 
	nQuantity:= 1, 
	nMBAddr:= 70, 
	cbLength:= SIZEOF(wInputRegsDigitalIn), 
	pDestAddr:= ADR(wInputRegsDigitalIn), 
	bExecute:= bSekvensFlagga AND bEnable, 
	tTimeout:= tTimeOut, 
	bBusy=> , 
	bError=> , 
	nErrId=> , 
	cbRead=> );
	
	DI1_V := wInputRegsDigitalIn.0;
	DI2_V := wInputRegsDigitalIn.1;
	DI3_V := wInputRegsDigitalIn.2;
	DI4_V := wInputRegsDigitalIn.3;
	DI5_V := wInputRegsDigitalIn.4;
	DI6_V := wInputRegsDigitalIn.5;
	DI7_V := wInputRegsDigitalIn.6;
	DI8_V := wInputRegsDigitalIn.7;
	DI9_V := wInputRegsDigitalIn.8;
	DI10_V := wInputRegsDigitalIn.9;
	DI11_V := wInputRegsDigitalIn.10;
	DI12_V := wInputRegsDigitalIn.11;
END_METHOD

METHOD PRIVATE mDigitalOut
VAR_INPUT
END_VAR
	CASE iStep OF

	0: 	//Start/reset
		bBusy := FALSE;
						
		IF bEnable AND bSekvensFlagga THEN
			iStep := 1;
			bError := FALSE;
		END_IF
		
	1: //Read Data (Value on output)
		bBusy := TRUE;
		FB_MBReadRegs_ArrHolding1.bExecute := TRUE;

		//Read Values
		FB_MBReadRegs_ArrHolding1(
			sIPAddr:= modbusTCP.sIpAddr, 
			nTCPPort:= modbusTCP.nTCPPort, 
			nUnitID:= nUnitID, 
			nQuantity:= 2, 
			nMBAddr:= 71, 
			cbLength:= SIZEOF(ArrHolding1), 
			pDestAddr:= ADR(ArrHolding1), 
			bExecute:=, 
			tTimeout:= tTimeOut, 
			bBusy=> ,
			bError=> , 
			nErrId=> , 
			cbRead=> );
	
		//Values
		DO1_V := ArrHolding1[0].0;
		DO2_V := ArrHolding1[0].1;
		DO3_V := ArrHolding1[0].2;
		DO4_V := ArrHolding1[0].3;
		TRANSISTOR_DO1_V := ArrHolding1[0].4;
		TRANSISTOR_DO2_V := ArrHolding1[0].5;
		TRANSISTOR_DO3_V := ArrHolding1[0].6;
		TRANSISTOR_DO4_V := ArrHolding1[0].7;

		//Error 
		IF FB_MBReadRegs_ArrHolding1.bError THEN
			FB_MBReadRegs_ArrHolding1(bExecute := FALSE);
			iStep := 99;
		END_IF
	
		//Gå till nästa steg
		IF NOT FB_MBReadRegs_ArrHolding1.bBusy AND NOT FB_MBReadRegs_ArrHolding1.bError THEN
			FB_MBReadRegs_ArrHolding1(bExecute := FALSE);
			bError := FALSE;
			iStep := 2;
		END_IF;

	2: //Read/Write communication error timedelay (config)
		bBusy := TRUE;

		//User input
		IF SP1 < 0 THEN
			SP1 := 0;
		END_IF;
		
		IF SP1 > 65535 THEN
			SP1 := 655;
		END_IF;
		
		fbReadWriteHoldingRegReal_ComError.bEnable := TRUE;
		
		fbReadWriteHoldingRegReal_ComError(
			sIPAddr:= modbusTCP.sIpAddr, 
			nTCPPort:= modbusTCP.nTCPPort, 
			nUnitID:= nUnitID, 
			mBusAdr:= 66, 
			bEnable:= , 
			tTimeout:= tTimeOut, 
			rReal:= SP1, 
			uiFaktor:= 100, 
			bError=> , 
			bBusy=> , 
			bSuccess=> );
				
		//Error 
		IF fbReadWriteHoldingRegReal_ComError.bError THEN
			fbReadWriteHoldingRegReal_ComError(bEnable := FALSE);
			iStep := 99;
		END_IF
	
		//Gå till nästa steg
		IF NOT fbReadWriteHoldingRegReal_ComError.bBusy AND NOT fbReadWriteHoldingRegReal_ComError.bError THEN
			fbReadWriteHoldingRegReal_ComError(bEnable := FALSE);
			bError := FALSE;
			iStep := 3;
		END_IF;
	
	3:	//Read/Write default values (config)
		//Config in IO
		wReadConfig.0 := ArrHolding1[1].0;
		wReadConfig.1 := ArrHolding1[1].1;
		wReadConfig.2 := ArrHolding1[1].2;
		wReadConfig.3 := ArrHolding1[1].3;
		wReadConfig.4 := ArrHolding1[1].4;
		wReadConfig.5 := ArrHolding1[1].5;
		wReadConfig.6 := ArrHolding1[1].6;
		wReadConfig.7 := ArrHolding1[1].7;
		//Config in PLC	
		wWriteConfig.0 := bDO1fallback; 
		wWriteConfig.1 := bDO2fallback;
		wWriteConfig.2 := bDO3fallback;
		wWriteConfig.3 := bDO4fallback;
		wWriteConfig.4 := bTransistorDO1fallback; 
		wWriteConfig.5 := bTransistorDO2fallback;
		wWriteConfig.6 := bTransistorDO3fallback;
		wWriteConfig.7 := bTransistorDO4fallback;
		
		bBusy := TRUE;	
		IF wReadConfig <> wWriteConfig THEN
			FB_MBWriteRegs_Config.bExecute := TRUE;
		END_IF
		
		FB_MBWriteRegs_Config(
			sIPAddr:= modbusTCP.sIpAddr, 
			nTCPPort:= modbusTCP.nTCPPort, 
			nUnitID:= nUnitID,
			nMBAddr:= 73,
			nValue:= wWriteConfig, 
			bExecute:= , 
			tTimeout:= tTimeout , 
			bBusy=> , 
			bError=> , 
			nErrId=> );
			
		IF FB_MBWriteRegs_Config.bError THEN
			FB_MBWriteRegs_Config(bExecute := FALSE);
			iStep := 99;
		END_IF
	
		//Next step
		IF NOT FB_MBWriteRegs_Config.bBusy AND NOT FB_MBWriteRegs_Config.bError THEN
			FB_MBWriteRegs_Config(bExecute := FALSE);
			bError := FALSE;
			iStep := 4;
		END_IF;

	4: //Write outputs
		bBusy := TRUE;	
			
		wWriteOutputs.0 := bDO1;
		wWriteOutputs.1 := bDO2;
		wWriteOutputs.2 := bDO3;
		wWriteOutputs.3 := bDO4;
		wWriteOutputs.4 := bTransistorDO1;
		wWriteOutputs.5 := bTransistorDO2;
		wWriteOutputs.6 := bTransistorDO3;
		wWriteOutputs.7 := bTransistorDO4;
		
		FB_MBWriteRegs_Outputs.bExecute := TRUE;
		
		FB_MBWriteRegs_Outputs(
			sIPAddr:= modbusTCP.sIpAddr, 
			nTCPPort:= modbusTCP.nTCPPort, 
			nUnitID:= nUnitID,
			nMBAddr:= 71,
			nValue:= wWriteOutputs, 
			bExecute:= , 
			tTimeout:= tTimeout , 
			bBusy=> , 
			bError=> , 
			nErrId=> );
				
		IF FB_MBWriteRegs_Outputs.bError THEN
			FB_MBWriteRegs_Outputs(bExecute := FALSE);
			iStep := 99;
		END_IF
	
		//Next step
		IF NOT FB_MBWriteRegs_Outputs.bBusy AND NOT FB_MBWriteRegs_Outputs.bError THEN
			FB_MBWriteRegs_Outputs(bExecute := FALSE);
			bError := FALSE;
			iStep := 20;
		END_IF;

	20: //Done
		bBusy := FALSE;
		iStep := 0;
		

	99: //Error handling
		bBusy := FALSE;
		bError := TRUE;
		iStep := 0;
		
END_CASE
END_METHOD

METHOD mRawToAnalog : REAL
VAR_INPUT
	rValueToConvert : WORD; //Rå-värde
END_VAR

VAR
	x1 : REAL;
	x2 : REAL;
	y1 : REAL;
	y2 : REAL;
	rTemp : REAL;
END_VAR
//0-10V
rTemp := fSignedConverter(rValueToConvert);

x1 := 0; 
x2 := 32767;
y1 := 0; 
y2 := 10.24; 
mRawToAnalog := fScale2p(rTemp, y1, y2, x1, x2);
END_METHOD

END_FUNCTION_BLOCK

// oaksModbusLibrary/Mitsubishi/fbMitsubishiATA_ATW
//OAKS AB
//2020-05-12
//Funktionsblock för kommunikation med en styrenhet för FLK från Mitshubishi via RS485 (via TCP/IP Gateway)
//Dubbelriktad modbusskrivning för börvärde
FUNCTION_BLOCK fbMitsubishiATA_ATW
VAR_INPUT
	sIPAddr : STRING := ''; 
	nTCPPort : UINT;
	nUnitID : UINT :=1;
	iModbusLoop : INT :=1; //Modbusslinga
	SP AT %M*  : REAL;//Börvärde~wp:[unit]°C[format]0.0[trendoption]i:300
				
END_VAR
VAR_OUTPUT
	
	V AT %M*  : BOOL;//Driftindikering~wp:[trendoptions]i:14400, t:1
	PV AT %M*  : REAL;//Rumstemperatur~wp:[unit]°C[format]0.0[trendoption]i:300
	PV1 AT %M*  : REAL;//Felkod (8000=Inget fel)~wp:[format]0
	PV6 AT %M*  : REAL;//Fläkthastighet~wp:[format]0
	PV7 AT %M*  : REAL;//Driftläge~wp:[format]0
	PV10 AT %M* : STRING;//Modbus konfiguering~wp:
	AL AT %M* : BOOL;//Summalarm~wp:
	FAULT AT %M* : BOOL;//Kommunikationsfel~wp:
	
END_VAR
VAR
	offset : WORD;
	rTemp : REAL;
	iTemp : UINT;
	bSekvensFlagga : BOOL;
			
	fbReadInputRegs_wInputRegs1: FB_MBReadInputRegs;
	wInputRegs1 : WORD; //Holding
		
	fbReadInputRegs_wInputRegs2: FB_MBReadInputRegs;
	wInputRegs2: WORD;
	
	fbReadRegs_wHolding1: FB_MBReadRegs;
	wArrayHolding1: ARRAY [1..13] OF WORD;
		
	//Kommunikationsfel
	fbKommTof : tof; 
	fbKommTon : ton;
	TON_alarm: TON;

	fbWriteHoldingDoubleControlled_Sp: fbDoubleControlledModbusHolding;
	
	sIP: STRING(255);
	sPort: STRING(255);
	sModbusID: STRING(255);
	sModbusLoop: STRING(255);
	
	sTemp: STRING(255);
END_VAR

//General
	offset := -1;
//Sekvens	
	bSekvensFlagga := oaksGVL.aBModbusSekvens[iModbusLoop] = UINT_TO_INT(nUnitID);
//Modbus konfiguering
	sIP := CONCAT (SIPAddr, '');
	sPort := CONCAT ('<br>Port: ', UINT_TO_STRING(nTCPPort)); 								
	sModbusID := CONCAT('<br>ID: ', UINT_TO_STRING(nUnitID));
	sModbusLoop := CONCAT('<br>Loop: ', INT_TO_STRING(iModbusLoop));

	sTemp := sIP;
	sTemp := CONCAT(sTemp, sPort);
	sTemp := CONCAT(sTemp, sModbusID);
	sTemp := CONCAT(sTemp, sModbusLoop);
		
	PV10 := sTemp;

///////////////		
//READ
///////////////		
	
//Read Inputregs 1
	//Roomtemp
	fbReadInputRegs_wInputRegs1(
	sIPAddr:= sIpAddr, 
	nTCPPort:= INT_TO_UINT(nTCPPort), 
	nUnitID:= INT_TO_BYTE(nUnitID), 
	nQuantity:= 1, 
	nMBAddr:= 1 + offset, 
	cbLength:= SIZEOF(wInputRegs1), 
	pDestAddr:= ADR(wInputRegs1), 
	bExecute:= bSekvensFlagga, 
	tTimeout:= T#3S, 
	bBusy=> , 
	bError=> , 
	nErrId=> , 
	cbRead=> );
	
	//Values
	PV := WORD_TO_REAL(wInputRegs1) / 10;
	
//Read Inputregs 2 
	//Error Code
	fbReadInputRegs_wInputRegs2(
	sIPAddr:= sIpAddr, 
	nTCPPort:= INT_TO_UINT(nTCPPort), 
	nUnitID:= INT_TO_BYTE(nUnitID), 
	nQuantity:= 1, 
	nMBAddr:= 9 + offset, 
	cbLength:= SIZEOF(wInputRegs2), 
	pDestAddr:= ADR(wInputRegs2), 
	bExecute:= bSekvensFlagga, 
	tTimeout:= T#3S, 
	bBusy=> , 
	bError=> , 
	nErrId=> , 
	cbRead=> );
	
	//Values
	PV1 := WORD_TO_REAL(wInputRegs2);
	
	//Error	
	TON_alarm(IN:= (PV1<>8000), PT:= T#1M , Q=> , ET=> );
	AL := TON_alarm.Q;

//Read Holding 1

	//Run
	fbReadRegs_wHolding1(
	sIPAddr:= sIpAddr, 
	nTCPPort:= INT_TO_UINT(nTCPPort), 
	nUnitID:= INT_TO_BYTE(nUnitID), 
	nQuantity:= 13, 
	nMBAddr:= 1 + offset, 
	cbLength:= SIZEOF(wArrayHolding1), 
	pDestAddr:= ADR(wArrayHolding1), 
	bExecute:= bSekvensFlagga, 
	tTimeout:= T#3S, 
	bBusy=> , 
	bError=> , 
	nErrId=> , 
	cbRead=> );
		
	PV6 := wArrayHolding1[1];
	wArrayHolding1[2];
	PV7 := wArrayHolding1[3];
	wArrayHolding1[4];
	wArrayHolding1[5];
	wArrayHolding1[6];
	wArrayHolding1[7];
	V := WORD_TO_BOOL(wArrayHolding1[8]);
	wArrayHolding1[9];
	wArrayHolding1[10];
	wArrayHolding1[11];
	wArrayHolding1[12];
	wArrayHolding1[13];

	
//		
//READ/WRITE Analogue registers		
//

	fbWriteHoldingDoubleControlled_Sp(
	sIPAddr:= sIPAddr, 
	nTCPPort:= nTCPPort, 
	nUnitID:= UINT_TO_BYTE(nUnitID) , 
	nMBAddr:= 2+offset, 
	bExecute:=bSekvensFlagga , 
	rScale:= 10, 
	rWrite:= SP, 
	bBusy=> , 
	bError=> );
	
//Communication error
	fbKommTof(IN:=fbReadInputRegs_wInputRegs1.bError , PT:=T#20S , Q=> , ET=> );
	fbKommTon(IN:=fbKommTof.Q , PT:=T#20M , Q=> , ET=> );
	FAULT :=fbKommTon.Q;
		
//Write busy	
	oaksgvl.aBModbusBusyFlagga[iModbusLoop,nUnitID] := fbReadInputRegs_wInputRegs1.bBusy OR fbReadInputRegs_wInputRegs2.bBusy OR fbWriteHoldingDoubleControlled_Sp.bBusy;

END_FUNCTION_BLOCK

// oaksModbusLibrary/Mitsubishi/fbMitsubishiHydroBox
//OAKS AB
//2020-07-06
//Funktionsblock för kommunikation med en styrenhet HydroBox. 
FUNCTION_BLOCK fbMitsubishiHydroBox
VAR_INPUT
	sIPAddr : STRING := ''; 
	nTCPPort : UINT;
	nUnitID : UINT :=1;
	iModbusLoop : INT :=1; //Modbusslinga
	bStart : BOOL; //Starta värmepump
	bCoolMode : BOOL; //Aktivera kylläge
	rSetpoint : REAL; //Börvärde värme/kyla
				
END_VAR
VAR_OUTPUT
	COMPRESSOR_V AT %M* : BOOL;//Driftindikering~wp:[trendoptions]i:14400, t:1
	COMPRESSOR_OP AT %M* : REAL;//Hastighet~wp:[unit]Hz[format]0[trendoptions]i:300
	PV1 AT %M* : STRING;//Drifläge~wp:[trendoptions]i:14400, t:1	
	SUPPLY_TEMPERATURE_PV AT %M* : REAL;//Utgående vattentemperatur~wp:[unit]°C[format]0.0[trendoptions]i:300
	RETURN_TEMPERATURE_PV AT %M* : REAL;//Ingående vattentemperatur~wp:[unit]°C[format]0.0[trendoptions]i:300
	PV4 AT %M* : REAL;//Utomhusgivare i utedel~wp:[unit]°C[format]0.0[trendoptions]i:300
		
	PV5 AT %M* : REAL;//Larmkod~wp:[format]0[trendoptions]i:300
	PV6 AT %M* : BOOL;//Elpatron 1~wp:[format]0[trendoptions]i:14400, t:1
	PV7 AT %M* : BOOL;//Elpatron 2~wp:[format]0[trendoptions]i:14400, t:1
	
	PV8 AT %M* : STRING;//Modbus konfiguering~wp:
	
	AL AT %M* : BOOL;//Summalarm~wp:
	FAULT AT %M* : BOOL;//Kommunikationsfel~wp:
	
END_VAR
VAR
	itemp2 : INT;
	iTemp : INT;
	rTemp : REAL;
	offset : INT;
	bSekvensFlagga : BOOL;
		
	FB_MBReadRegs_Coils1: FB_MBReadInputs;
	coils1 : BYTE; //Holding	
 
	fbReadInputRegs_wReadRegs1alarm: FB_MBReadRegs;
	wrReadRegs1alarm: WORD;
	TON_alarm: TON;
	
	FB_MBReadRegs_ArrInputRegs1: FB_MBReadInputRegs;
	arrInputRegs1 : ARRAY [0..10] OF WORD; //Input registers
	
	FB_MBReadRegs_ArrHolding1: FB_MBReadRegs;
	ArrHolding1 : ARRAY [0..10] OF WORD; //Holding
	
	fbReadWriteHoldingReg_1: fbReadWriteHoldingReg;
	wWriteHolding1 : WORD;
	
	fbReadWriteHoldingReg_2: fbReadWriteHoldingReg;
	wWriteHolding2 : WORD;
	
	fbReadWriteHoldingReg_3: fbReadWriteHoldingReg;
	wWriteHolding3 : WORD;
	
	//Kommunikationsfel
	fbKommTof : tof; 
	fbKommTon : ton;
	
	//Modbus config
	sIP: STRING(255);
	sPort: STRING(255);
	sModbusID: STRING(255);
	sModbusLoop: STRING(255);
	sTemp : STRING(255);
		
	
	
END_VAR

//General
	offset := -1;
//Sekvens	
	bSekvensFlagga := oaksGVL.aBModbusSekvens[iModbusLoop] = UINT_TO_INT(nUnitID);
//Modbus konfiguering
	sIP := CONCAT (SIPAddr, '');
	sPort := CONCAT ('<br>Port: ', UINT_TO_STRING(nTCPPort)); 								
	sModbusID := CONCAT('<br>ID: ', UINT_TO_STRING(nUnitID));
	sModbusLoop := CONCAT('<br>Loop: ', INT_TO_STRING(iModbusLoop));	

	sTemp := sIP;
	sTemp := CONCAT(sTemp, sPort);
	sTemp := CONCAT(sTemp, sModbusID);
	sTemp := CONCAT(sTemp, sModbusLoop);
	
	PV8 := sTemp;

///////////////		
//READ
///////////////

//COILS

	FB_MBReadRegs_Coils1(
	sIPAddr:= sIpAddr, 
	nTCPPort:= INT_TO_UINT(nTCPPort), 
	nUnitID:= INT_TO_BYTE(nUnitID), 
	nQuantity:= 2, 
	nMBAddr:= 18 + offset, 
	cbLength:= SIZEOF(coils1), 
	pDestAddr:= ADR(coils1), 
	bExecute:= bSekvensFlagga, 
	tTimeout:= T#3S, 
	bBusy=> , 
	bError=> , 
	nErrId=> , 
	cbRead=> );		

		//Values
		PV6 := coils1.0; //0
		PV7 := coils1.1; //1		

//INPUT REGISTERS		
		
//Read Inputregs 1 (Alarm)
	//Error Code
	fbReadInputRegs_wReadRegs1alarm(
	sIPAddr:= sIpAddr, 
	nTCPPort:= INT_TO_UINT(nTCPPort), 
	nUnitID:= INT_TO_BYTE(nUnitID), 
	nQuantity:= 1, 
	nMBAddr:= 13 + offset, 
	cbLength:= SIZEOF(wrReadRegs1alarm), 
	pDestAddr:= ADR(wrReadRegs1alarm), 
	bExecute:= bSekvensFlagga, 
	tTimeout:= T#3S, 
	bBusy=> , 
	bError=> , 
	nErrId=> , 
	cbRead=> );
	
	//Values
	PV5 := WORD_TO_REAL(wrReadRegs1alarm);
	
	//Error	
	TON_alarm(IN:= (PV5<>8000), PT:= T#1M , Q=> , ET=> );
	AL := TON_alarm.Q;		

	//Read input registers 59-63
	FB_MBReadRegs_ArrInputRegs1(
	sIPAddr:= sIpAddr, 
	nTCPPort:= INT_TO_UINT(nTCPPort), 
	nUnitID:= INT_TO_BYTE(nUnitID), 
	nQuantity:= 5, 
	nMBAddr:= 59 + offset, 
	cbLength:= SIZEOF(arrInputRegs1), 
	pDestAddr:= ADR(arrInputRegs1), 
	bExecute:= bSekvensFlagga, 
	tTimeout:= T#3S, 
	bBusy=> , 
	bError=> , 
	nErrId=> , 
	cbRead=> );
		//Values
		rTemp := WORD_TO_REAL(arrInputRegs1[0]); //59
		PV4 := fSignedConverter(rInput:=rTemp ) / 10;
		//arrInputRegs1[1]; //60
		SUPPLY_TEMPERATURE_PV := WORD_TO_REAL(arrInputRegs1[2]) / 100; //61
		//arrInputRegs1[3]; //62
		RETURN_TEMPERATURE_PV := WORD_TO_REAL(arrInputRegs1[4]) / 100; //63
		//arrInputRegs1[5]; //5
		//arrInputRegs1[6]; //6
		//arrInputRegs1[7]; //7
		//arrInputRegs1[8]; //8
		//arrInputRegs1[9]; //9
		//arrInputRegs1[10]; //10

//HOLDING	
	
	//Read Holding 74 (mode)
	FB_MBReadRegs_ArrHolding1(
	sIPAddr:= sIpAddr, 
	nTCPPort:= INT_TO_UINT(nTCPPort), 
	nUnitID:= INT_TO_BYTE(nUnitID), 
	nQuantity:= 1, 
	nMBAddr:= 74 + offset, 
	cbLength:= SIZEOF(ArrHolding1), 
	pDestAddr:= ADR(ArrHolding1), 
	bExecute:= bSekvensFlagga, 
	tTimeout:= T#3S, 
	bBusy=> , 
	bError=> , 
	nErrId=> , 
	cbRead=> );
	
		//Values
		COMPRESSOR_OP := WORD_TO_REAL(ArrHolding1[0]); //0
		COMPRESSOR_V := COMPRESSOR_OP > 0;
		//ArrHolding1[1]; //1
		//ArrHolding1[2]; //2
		//ArrHolding1[3]; //3
		//ArrHolding1[4]; //4
		//ArrHolding1[5]; //5
		//ArrHolding1[6]; //6
		//ArrHolding1[7]; //7
		//ArrHolding1[8]; //8
		//ArrHolding1[9]; //9
		//ArrHolding1[10]; //10

//HOLDING READ/WRITE

	//Read/Write holding (start)
	//0=Av, 1=På
	IF bStart THEN
		wWriteHolding1 := 1;
	ELSE 
		wWriteHolding1 := 0;
	
	END_IF
	
	fbReadWriteHoldingReg_1(
	sIPAddr:= sIpAddr, 
	nTCPPort:= INT_TO_UINT(nTCPPort), 
	nUnitID:= INT_TO_BYTE(nUnitID), 
	mBusAdr:= 26 + offset, 
	bEnable:= bSekvensFlagga, 
	iWrite:= wWriteHolding1, 
	iRead=> , 
	bError=> , 
	bBusy=> );

	//Read/Write holding (heat/cool)
	//1=Värmeläge, 4=kylläge
	IF bCoolMode THEN
		wWriteHolding2 := 4;
		PV1 := 'Kyla';
	ELSE 
		wWriteHolding2 := 1;
		PV1 := 'Värme';
	END_IF
	
	fbReadWriteHoldingReg_2(
	sIPAddr:= sIpAddr, 
	nTCPPort:= INT_TO_UINT(nTCPPort), 
	nUnitID:= INT_TO_BYTE(nUnitID), 
	mBusAdr:= 29 + offset, 
	bEnable:= bSekvensFlagga, 
	iWrite:= wWriteHolding2, 
	iRead=> , 
	bError=> , 
	bBusy=> );
		
	//Read/Write holding (setpoint)
	iTemp := REAL_TO_INT(rSetpoint) * 100;
		
	fbReadWriteHoldingReg_3(
	sIPAddr:= sIpAddr, 
	nTCPPort:= INT_TO_UINT(nTCPPort), 
	nUnitID:= INT_TO_BYTE(nUnitID), 
	mBusAdr:= 33 + offset, 
	bEnable:= bSekvensFlagga, 
	iWrite:= INT_TO_WORD(iTemp), 
	iRead=> , 
	bError=> , 
	bBusy=> );				
	
//Communication error
	fbKommTof(IN:= 	FB_MBReadRegs_Coils1.bError OR
	fbReadInputRegs_wReadRegs1alarm.bError OR
	FB_MBReadRegs_ArrInputRegs1.bError OR
	FB_MBReadRegs_ArrHolding1.bError OR
	fbReadWriteHoldingReg_1.bError OR
	fbReadWriteHoldingReg_2.bError OR
	fbReadWriteHoldingReg_3.bError, 
	PT:=T#20S , Q=> , ET=> );
	fbKommTon(IN:=fbKommTof.Q , PT:=T#20M , Q=> , ET=> );
	FAULT :=fbKommTon.Q;
		
//Write busy	
	oaksgvl.aBModbusBusyFlagga[iModbusLoop,nUnitID] := 
	FB_MBReadRegs_Coils1.bBusy OR
	fbReadInputRegs_wReadRegs1alarm.bBusy OR
	FB_MBReadRegs_ArrInputRegs1.bBusy OR
	FB_MBReadRegs_ArrHolding1.bBusy OR
	fbReadWriteHoldingReg_1.bBusy OR
	fbReadWriteHoldingReg_2.bBusy OR
	fbReadWriteHoldingReg_3.bBusy;

END_FUNCTION_BLOCK

// oaksModbusLibrary/Nicotra Gebhardt/fbNicotraGebhardtRLM
//OAKS AB
//2022-10-31
//Ver. 1.0
//Modbusblock för Nicotra Gebhardt RLM fläkt.
FUNCTION_BLOCK fbNicotraGebhardtRLM
VAR_INPUT
	sIPAddr : STRING := ''; 
	nTCPPort : UINT;
	nUnitID : UINT :=1;
	iModbusLoop : INT :=1; //Modbusslinga
			
END_VAR
VAR_OUTPUT
	RPM AT %M* : REAL;//Varvtal~wp:[unit]RPM[format]0[trendoptions]i:300
	U1 AT %M* : REAL;//Spänning~wp:[unit]V[format]0[trendoptions]i:300
	I1 AT %M* : REAL;//Ampere~wp:[unit]A[format]0.0[trendoptions]i:300	
	P1 AT %M* : REAL;//Effekt~wp:[unit]kW[format]0.0[trendoptions]i:300	
	E1 AT %M* : REAL;//Energi~wp:[unit]kWh[format]0.0[trendoptions]i:300		
	PV8 AT %M* : STRING;//Modbus konfiguering~wp:
	FAULT AT %M* : BOOL;//Kommunikationsfel~wp:[alarmoptions]p:2
	
END_VAR
VAR
	offset : UINT;
	rTemp1 : REAL;	
	rTemp2 : REAL;	
	rTemp3 : REAL;	
	bSekvensFlagga : BOOL;
			
	FB_MBReadRegs_ArrReadInputsRegs1 : FB_MBReadInputRegs;	
	wArrReadInputsRegs1 : ARRAY [0..33] OF WORD; //ReadInputsRegs
		
	//Kommunikationsfel
	fbKommTof : tof; 
	fbKommTon : fbAlarm;
	
	sIP: STRING(255);
	sPort: STRING(255);
	sModbusID: STRING(255);
	sModbusLoop: STRING(255);
	sTemp : STRING(255);
	
END_VAR

//General
	offset := 0;
//Sekvens	
	bSekvensFlagga := oaksGVL.aBModbusSekvens[iModbusLoop] = UINT_TO_INT(nUnitID);
//Modbus konfiguering
	sIP := CONCAT (SIPAddr, '');
	sPort := CONCAT ('<br>Port: ', UINT_TO_STRING(nTCPPort)); 								
	sModbusID := CONCAT('<br>ID: ', UINT_TO_STRING(nUnitID));
	sModbusLoop := CONCAT('<br>Loop: ', INT_TO_STRING(iModbusLoop));	

	sTemp := sIP;
	sTemp := CONCAT(sTemp, sPort);
	sTemp := CONCAT(sTemp, sModbusID);
	sTemp := CONCAT(sTemp, sModbusLoop);
	
	PV8 := sTemp;

///////////////		
//READ
///////////////		
	
	//Read Inputs 0-33
	FB_MBReadRegs_ArrReadInputsRegs1(
	sIPAddr:= sIpAddr, 
	nTCPPort:= (nTCPPort), 
	nUnitID:= UINT_TO_BYTE(nUnitID), 
	nQuantity:= 34, 
	nMBAddr:= 0 + offset,
	cbLength:= SIZEOF(wArrReadInputsRegs1), 
	pDestAddr:= ADR(wArrReadInputsRegs1), 
	bExecute:= bSekvensFlagga,
	tTimeout:= T#10S, 
	bBusy=> , 
	bError=> , 
	nErrId=> , 
	cbRead=> );	
	
		//Values
		//wArrReadInputsRegs1[0]; //0 - Drive Type, Res.:1, Unit:-
		//wArrReadInputsRegs1[1]; //1 - AOC SW version, Res.:0.01, Unit:-
		//wArrReadInputsRegs1[2]; //2 - MOC SW version, Res.:0.01, Unit:-
		//wArrReadInputsRegs1[3]; //3 - PrcOut, Res.:0.01, Unit:%
		RPM := wArrReadInputsRegs1[4]; //4 - RPMOut, (PM) Res.:1, Unit:RPM or (AC)Res.:0.01, Unit:Hz
		//wArrReadInputsRegs1[5]; //5 - Intern Temp, Res.:0.01, Unit:ºC
		//wArrReadInputsRegs1[6]; //6 - V In (RMS), Res.:1, Unit:V
		I1 := (wArrReadInputsRegs1[7]*0.001); //7 - I Out, Res.:0.01, Unit:A
		P1 := wArrReadInputsRegs1[8]*0.001; //8 - Power In (filtered), Res.:0.01, Unit:kW
		//wArrReadInputsRegs1[9]*1000; //9 - I Ripple, Res.:0.01, Unit:A
	
		//wArrReadInputsRegs1[10]; //10 - Operation Minutes, Res.:1, Unit:Min
		//wArrReadInputsRegs1[11]; //11 - Operation Day, Res.:1, Unit:Day
		//wArrReadInputsRegs1[12]; //12 - V Ripple, Res.:1, Unit:V
		//wArrReadInputsRegs1[13]; //13 - Config file variant, 2 ASCII characters
		//wArrReadInputsRegs1[14]; //14 - Config file version, Res.:0.01, Unit:-
		//wArrReadInputsRegs1[15]; //15 - ExternSet, Res.:1, Unit:mV
		//wArrReadInputsRegs1[16]; //16 - Power Supply, Res.:1, Unit:V
		//wArrReadInputsRegs1[17]; //17 - OverVoltageCount, Res.:1, Unit:-
		//wArrReadInputsRegs1[18]; //18 - AOC SW variant, Res.:-, Unit:-
		//wArrReadInputsRegs1[19]; //19 - AOC Boot SW, Res.:0.01, Unit:-

		//wArrReadInputsRegs1[20]; //20 - MOC Boot SW, Res.:0.01, Unit:-
		//wArrReadInputsRegs1[21]; //21 - Motor Cfg. Var, Res.:1, Unit:-
		//wArrReadInputsRegs1[22]; //22 - Motor Cfg. Ver., Res.:0.01, Unit:-
		//wArrReadInputsRegs1[23]; //23 - Fan Cfg. Var., Res.:1, Unit:-
		//wArrReadInputsRegs1[24]; //24 - Fan Cfg. Ver, Res.:0.01, Unit:-
		//wArrReadInputsRegs1[25]; //25 - User Data Var., Res.:1, Unit:-
		//wArrReadInputsRegs1[26]; //26 - User Data Ver, Res.:0.01, Unit:-
		//wArrReadInputsRegs1[27]; //27 - IOM SW version, Res.:0.01, Unit:-
		//wArrReadInputsRegs1[28]; //28 - V DC Bus (Peak).:1, Unit:V
		U1 := wArrReadInputsRegs1[29]; //29 - V Motor (Peak), Res.:1, Unit:V

		//wArrReadInputsRegs1[30]*1000; //0 - Power In (unfilterd), Res.:0.01, Unit:kW
		rTemp1 := WORD_TO_REAL (wArrReadInputsRegs1[31]); //1 - Power Consumpt., Res.:1, Unit:Wh
		rTemp2 := WORD_TO_REAL (wArrReadInputsRegs1[32]); //2 - Power Consumpt., Res.:1, Unit:kWh
		rTemp3 := WORD_TO_REAL (wArrReadInputsRegs1[33]); //3 - Power Consumpt., Res.:1, Unit:MWh
		E1 := (((rTemp3 * 1000000) + (rTemp2 * 1000) + rTemp1)*0.001);
	
//Communication error
	fbKommTof(IN:=FB_MBReadRegs_ArrReadInputsRegs1.bError , PT:=T#60S , Q=> , ET=> );
	fbKommTon(bInput:=fbKommTof.Q , tAlarmDelay:=T#20M , bAutoReset:= , bAlarmOutput=> );
	FAULT :=fbKommTon.bAlarmOutput;
		
//Write busy	
	oaksgvl.aBModbusBusyFlagga[iModbusLoop,nUnitID] := FB_MBReadRegs_ArrReadInputsRegs1.bBusy;

END_FUNCTION_BLOCK

// oaksModbusLibrary/Produal/Givare/fbProdualHdhmCo2
//OAKS AB
//2020-03-17
//Funktionsblock för modbus-TCP, Produal HDK-M Koldioxid/temp-givare

FUNCTION_BLOCK fbProdualHdhmCo2
VAR_INPUT
	sIPAddr : STRING := ''; 
	nTCPPort : UINT;
	nUnitID : UINT;
	iModbusLoop : INT :=1; //Modbusslinga
	
END_VAR
VAR_OUTPUT
	PV AT %M*: REAL; //Temperatur~wp:[unit]°C[format]0.0[trendoptions]i:300
	PV1 AT %M* : REAL; //Koldioxidhalt~wp:[unit]ppm[format]0[trendoptions]i:300
	FAULT AT %M*: BOOL; //Kommunikationsfel~wp:
	PV8 AT %M* : STRING;//Modbus konfiguering~wp:
END_VAR
VAR
	
	sIP: STRING(255);
	sPort: STRING(255);
	sModbusID: STRING(255);
	sModbusLoop: STRING(255);
	sTemp : STRING(255);
	iTemp : UINT;
	fbKommTof : tof; 
	fbKommTon : ton;
	fbTempCo2: FB_MBReadInputRegs;
	wTempCo2 : ARRAY[0..1] OF	WORD; 
	bSekvensFlagga : BOOL;
END_VAR
VAR_INPUT PERSISTENT
	rCalTemp : REAL;
	rCalCo2 : REAL;
END_VAR

//Modbus konfiguering
	sIP := CONCAT (SIPAddr, '');
	sPort := CONCAT ('<br>Port: ', UINT_TO_STRING(nTCPPort)); 								
	sModbusID := CONCAT('<br>ID: ', UINT_TO_STRING(nUnitID));
	sModbusLoop := CONCAT('<br>Loop: ', INT_TO_STRING(iModbusLoop));	

	sTemp := sIP;
	sTemp := CONCAT(sTemp, sPort);
	sTemp := CONCAT(sTemp, sModbusID);
	sTemp := CONCAT(sTemp, sModbusLoop);
	
	PV8 := sTemp;

//Sekvens	
	bSekvensFlagga := oaksGVL.aBModbusSekvens[iModbusLoop] = UINT_TO_INT(nUnitID);
	
	fbTempCo2(
	sIPAddr:= sIpAddr, 
	nTCPPort:= INT_TO_UINT(nTCPPort), 
	nUnitID:= INT_TO_BYTE(nUnitID), 
	nQuantity:=2 , 
	nMBAddr:=0 , 
	cbLength:= SIZEOF(wTempCo2), 
	pDestAddr:= ADR(wTempCo2), 
	bExecute:= bSekvensFlagga, 
	tTimeout:= T#20S, 
	bBusy=> , 
	bError=> , 
	nErrId=> , 
	cbRead=> );
	
	fbKommTof(IN:=fbTempCo2.bError , PT:=T#20S , Q=> , ET=> );
	fbKommTon(IN:=fbKommTof.Q , PT:=T#20M , Q=> , ET=> );
	FAULT :=fbKommTon.Q;
	
	//Temp
	iTemp := WORD_TO_UINT(wTempCo2[1]);
	PV := (UINT_TO_REAL(iTemp) /10) + rCalTemp;
	
	//Co2
	iTemp := WORD_TO_UINT(wTempCo2[0]);
	PV1 := (UINT_TO_REAL(iTemp)) + rCalCo2;
	
	//Write busy	
	oaksgvl.aBModbusBusyFlagga[iModbusLoop,nUnitID] := fbTempCo2.bBusy;

END_FUNCTION_BLOCK

// oaksModbusLibrary/Produal/Givare/fbProdualHdhmPirCo2
//OAKS AB
//2021-11-29
//Funktionsblock för modbus-TCP, Produal HDK-M-PIR Koldioxid/temp-givare med inbyggd närvarogivare

FUNCTION_BLOCK fbProdualHdhmPirCo2
VAR_INPUT
	sIPAddr : STRING := ''; 
	nTCPPort : UINT;
	nUnitID : UINT;
	iModbusLoop : INT :=1; //Modbusslinga
	
END_VAR
VAR_OUTPUT
	V AT %M*: BOOL; //Närvaroindikering (fördröjt till och frånslag)~wp:[trendoptions]i:14400, t:1
	PV4 AT %M*: BOOL; //Närvarogivare~wp:[trendoptions]i:14400, t:1
	PV AT %M*: REAL; //Temperatur~wp:[unit]°C[format]0.0[trendoptions]i:300
	PV1 AT %M* : REAL; //Koldioxidhalt~wp:[unit]ppm[format]0[trendoptions]i:300
	FAULT AT %M*: BOOL; //Kommunikationsfel~wp:
	PV8 AT %M* : STRING;//Modbus konfiguering~wp:
END_VAR
VAR
	sIP: STRING(255);
	sPort: STRING(255);
	sModbusID: STRING(255);
	sModbusLoop: STRING(255);
	sTemp : STRING(255);
	iTemp : UINT;
	fbKommTof : tof; 
	fbKommTon : ton;
	fbTempCo2: FB_MBReadInputRegs;
	wTempCo2 : ARRAY[0..1] OF	WORD; 
	bSekvensFlagga : BOOL;
	
	uiStartDelay : UINT;
	uiStopDelay : UINT;
	
	fbWriteStartDelay : fbReadWriteHoldingReg;
	fbWriteStopDelay : fbReadWriteHoldingReg;
	
	fbReadPir : FB_MBReadInputs;
	
	bReadPir : BYTE; // 10002 PIR sensor state (immediate) - 10003 PIR sensor state (control)
END_VAR
VAR_INPUT PERSISTENT
	rCalTemp : REAL;
	rCalCo2 : REAL;
END_VAR
VAR PERSISTENT
	SP7 AT %M*: REAL; //Fördröjning aktivering närvaroindikering (0-1-2)~wp:[format]0
	SP8 AT %M*: REAL; //Fördröjning inaktivering närvaroindikering (0-1-2-3-4-5)~wp:[format]0
END_VAR

	IF SP7 <> 0 AND SP7 <> 1 AND SP7 <> 2 THEN // Kollar om inställning är inom tillåten intervall.
		SP7 := 1;
	ELSE
		uiStartDelay := fRealToWord(SP7,1);
	END_IF
	
	IF SP8 <> 0 AND SP8 <> 1 AND SP8 <> 2 AND SP8 <> 3 AND SP8 <> 4 AND SP8 <> 5 THEN // Kollar om inställning är inom tillåten intervall.
		SP8 := 3;
	ELSE
		uiStopDelay := fRealToWord(SP8,1);
	END_IF
	
	fbWriteStartDelay(
	sIPAddr:= sIpAddr, 
	nTCPPort:= INT_TO_UINT(nTCPPort), 
	nUnitID:= INT_TO_BYTE(nUnitID), 
	mBusAdr:=34 , 
	bEnable:=bSekvensFlagga , 
	iWrite:=uiStartDelay , 
	tTimeout:= T#20S , 
	iRead=> , 
	bError=> , 
	bBusy=> );  
	
	fbWriteStopDelay(
	sIPAddr:= sIpAddr, 
	nTCPPort:= INT_TO_UINT(nTCPPort), 
	nUnitID:= INT_TO_BYTE(nUnitID), 
	mBusAdr:=35 , 
	bEnable:=bSekvensFlagga , 
	iWrite:=uiStartDelay , 
	tTimeout:= T#20S , 
	iRead=> , 
	bError=> , 
	bBusy=> );
	
	fbReadPir(
	sIPAddr:= sIpAddr, 
	nTCPPort:= INT_TO_UINT(nTCPPort), 
	nUnitID:= INT_TO_BYTE(nUnitID), 
	nQuantity:= 2, 
	nMBAddr:= 1, 
	cbLength:= SIZEOF(bReadPir), 
	pDestAddr:= ADR(bReadPir), 
	bExecute:= bSekvensFlagga, 
	tTimeout:=T#20S , 
	bBusy=> , 
	bError=> , 
	nErrId=> , 
	cbRead=> );
	
	PV4 :=  bReadPir.0;
	V := bReadPir.1;
	

//Modbus konfiguering
	sIP := CONCAT (SIPAddr, '');
	sPort := CONCAT ('<br>Port: ', UINT_TO_STRING(nTCPPort)); 								
	sModbusID := CONCAT('<br>ID: ', UINT_TO_STRING(nUnitID));
	sModbusLoop := CONCAT('<br>Loop: ', INT_TO_STRING(iModbusLoop));	

	sTemp := sIP;
	sTemp := CONCAT(sTemp, sPort);
	sTemp := CONCAT(sTemp, sModbusID);
	sTemp := CONCAT(sTemp, sModbusLoop);
	
	PV8 := sTemp;

//Sekvens	
	bSekvensFlagga := oaksGVL.aBModbusSekvens[iModbusLoop] = UINT_TO_INT(nUnitID);
	
	fbTempCo2(
	sIPAddr:= sIpAddr, 
	nTCPPort:= INT_TO_UINT(nTCPPort), 
	nUnitID:= INT_TO_BYTE(nUnitID), 
	nQuantity:=2 , 
	nMBAddr:=0 , 
	cbLength:= SIZEOF(wTempCo2), 
	pDestAddr:= ADR(wTempCo2), 
	bExecute:= bSekvensFlagga, 
	tTimeout:= T#20S, 
	bBusy=> , 
	bError=> , 
	nErrId=> , 
	cbRead=> );
	
	fbKommTof(IN:=fbTempCo2.bError , PT:=T#20S , Q=> , ET=> );
	fbKommTon(IN:=fbKommTof.Q , PT:=T#20M , Q=> , ET=> );
	FAULT :=fbKommTon.Q;
	
	//Temp
	iTemp := WORD_TO_UINT(wTempCo2[1]);
	PV := (UINT_TO_REAL(iTemp) /10) + rCalTemp;
	
	//Co2
	iTemp := WORD_TO_UINT(wTempCo2[0]);
	PV1 := (UINT_TO_REAL(iTemp)) + rCalCo2;
	
	//Write busy	
	oaksgvl.aBModbusBusyFlagga[iModbusLoop,nUnitID] := fbTempCo2.bBusy;

END_FUNCTION_BLOCK

// oaksModbusLibrary/Produal/Givare/fbProdualHdhmTempCo2
FUNCTION_BLOCK fbProdualHdhmTempCo2
VAR_INPUT
	sIPAddr : STRING := ''; 
	nTCPPort : UINT;
	nUnitID : UINT;
	iModbusLoop : INT :=1; //Modbusslinga
	
END_VAR
VAR_OUTPUT
	rTemperature : REAL; // Temperatur
	rCo2 : REAL; // co2-halt
	rHumidity : REAL;  // fukthalt
	bFault : BOOL; // Kommunikationsfel
END_VAR
VAR
	fbKommTof : tof; 
	fbKommTon : ton;
	fbTempCo2Humidity: FB_MBReadInputRegs;
	wTempCo2Humidity : ARRAY[0..2] OF	WORD; 
	bSekvensFlagga : BOOL;
END_VAR

//Sekvens	
	bSekvensFlagga := oaksGVL.aBModbusSekvens[iModbusLoop] = UINT_TO_INT(nUnitID);
	
	fbTempCo2Humidity(
	sIPAddr:= sIpAddr, 
	nTCPPort:= INT_TO_UINT(nTCPPort), 
	nUnitID:= INT_TO_BYTE(nUnitID), 
	nQuantity:=3 , 
	nMBAddr:=0 , 
	cbLength:= SIZEOF(wTempCo2Humidity), 
	pDestAddr:= ADR(wTempCo2Humidity), 
	bExecute:= bSekvensFlagga, 
	tTimeout:= T#20S, 
	bBusy=> , 
	bError=> , 
	nErrId=> , 
	cbRead=> );
	
	fbKommTof(IN:=fbTempCo2Humidity.bError , PT:=T#20S , Q=> , ET=> );
	fbKommTon(IN:=fbKommTof.Q , PT:=T#20M , Q=> , ET=> );
	bFault :=fbKommTon.Q;
	
	rTemperature := wTempCo2Humidity[1] *0.1;
	rCo2 := wTempCo2Humidity[0];
	rHumidity := wTempCo2Humidity[2];
	
	//Write busy	
	oaksgvl.aBModbusBusyFlagga[iModbusLoop,nUnitID] := fbTempCo2Humidity.bBusy;

END_FUNCTION_BLOCK

// oaksModbusLibrary/Produal/Givare/fbProdualKLH
//OAKS AB
//2020-06-07
//Funktionsblock för modbus-TCP, Produal KLH Temperatur-/fuktgivare
FUNCTION_BLOCK fbProdualKLH
VAR_INPUT
	sIPAddr : STRING := ''; 
	nTCPPort : UINT;
	nUnitID : UINT;
	iModbusLoop : INT :=1; //Modbusslinga
	
END_VAR
VAR_OUTPUT
	PV AT %M*: REAL; //Temperatur~wp:[unit]°C[format]0.0[trendoptions]i:300
	PV1 AT %M* : REAL; //Fukthalt~wp:[unit]rH%[format]0[trendoptions]i:300
	FAULT AT %M*: BOOL; //Kommunikationsfel~wp:
	PV8 AT %M* : STRING;//Modbus konfiguering~wp:
END_VAR
VAR
	
	sIP: STRING(255);
	sPort: STRING(255);
	sModbusID: STRING(255);
	sModbusLoop: STRING(255);
	sTemp : STRING(255);
	rTemp : REAL;
	fbKommTof : tof; 
	fbKommTon : ton;
	fbTempHumidity: FB_MBReadInputRegs;
	wTempHumidity : ARRAY[1..2] OF	WORD; 
	bSekvensFlagga : BOOL;

END_VAR
VAR_INPUT PERSISTENT
	rCalTemp : REAL;
	rCalHumidity : REAL;
END_VAR

//Modbus konfiguering
	sIP := CONCAT (SIPAddr, '');
	sPort := CONCAT ('<br>Port: ', UINT_TO_STRING(nTCPPort)); 								
	sModbusID := CONCAT('<br>ID: ', UINT_TO_STRING(nUnitID));
	sModbusLoop := CONCAT('<br>Loop: ', INT_TO_STRING(iModbusLoop));	

	sTemp := sIP;
	sTemp := CONCAT(sTemp, sPort);
	sTemp := CONCAT(sTemp, sModbusID);
	sTemp := CONCAT(sTemp, sModbusLoop);
	
	PV8 := sTemp;

//Sekvens	
	bSekvensFlagga := oaksGVL.aBModbusSekvens[iModbusLoop] = UINT_TO_INT(nUnitID);
	
	fbTempHumidity(
	sIPAddr:= sIpAddr, 
	nTCPPort:= INT_TO_UINT(nTCPPort), 
	nUnitID:= INT_TO_BYTE(nUnitID), 
	nQuantity:=2 , 
	nMBAddr:=1 , 
	cbLength:= SIZEOF(wTempHumidity), 
	pDestAddr:= ADR(wTempHumidity), 
	bExecute:= bSekvensFlagga, 
	tTimeout:= T#20S, 
	bBusy=> , 
	bError=> , 
	nErrId=> , 
	cbRead=> );
	
	fbKommTof(IN:=fbTempHumidity.bError , PT:=T#20S , Q=> , ET=> );
	fbKommTon(IN:=fbKommTof.Q , PT:=T#20M , Q=> , ET=> );
	FAULT :=fbKommTon.Q;
	
	//Temp
	rTemp := fSignedConverter(rInput:= WORD_TO_REAL(wTempHumidity[1]));
	PV := (rTemp / 10) + rCalTemp;
	
	//Fukt
	rTemp := fSignedConverter(rInput:= WORD_TO_REAL(wTempHumidity[2]));
	PV1 := rTemp + rCalHumidity;
	
	//Write busy	
	oaksgvl.aBModbusBusyFlagga[iModbusLoop,nUnitID] := fbTempHumidity.bBusy;

END_FUNCTION_BLOCK

// oaksModbusLibrary/Produal/Givare/fbProdualPEL2500Mx
//OAKS AB
//2020-03-17
//Funktionsblock för modbus-TCP, Produal PEL2500-M (-N), tryckgivare med eller utan display.

FUNCTION_BLOCK fbProdualPEL2500Mx
VAR_INPUT
	sIPAddr : STRING := ''; 
	nTCPPort : UINT;
	nUnitID : UINT;
	iModbusLoop : INT :=1; //Modbusslinga
	
END_VAR
VAR_OUTPUT
	PV AT %M*: REAL; //Tryck~wp:[unit]Pa[format]0[trendoptions]i:300
	FAULT AT %M*: BOOL; //Kommunikationsfel~wp:
	PV8 AT %M* : STRING;//Modbus konfiguering~wp:
	PV9 AT %M* : UINT; //Tidskonstant~wp:
	PV10 AT %M* : STRING; //Konfigurering~wp:
	PV11 AT %M* : REAL; //Utsignal inom mätområde (0-100%)~wp:[unit]%[format]0.0
END_VAR
VAR
	sIP: STRING(255);
	sPort: STRING(255);
	sModbusID: STRING(255);
	sModbusLoop: STRING(255);
	sTemp : STRING(255);
	iTemp : UINT;
	fbKommTof : tof; 
	fbKommTon : ton;
	fbTempPress: FB_MBReadInputRegs;
	wArray1 : ARRAY[1..4] OF	WORD; 
	bSekvensFlagga : BOOL;
	rTemp : REAL;
END_VAR
VAR_INPUT PERSISTENT
	
END_VAR

//Modbus konfiguering
	sIP := CONCAT (SIPAddr, '');
	sPort := CONCAT ('<br>Port: ', UINT_TO_STRING(nTCPPort)); 								
	sModbusID := CONCAT('<br>ID: ', UINT_TO_STRING(nUnitID));
	sModbusLoop := CONCAT('<br>Loop: ', INT_TO_STRING(iModbusLoop));	

	sTemp := sIP;
	sTemp := CONCAT(sTemp, sPort);
	sTemp := CONCAT(sTemp, sModbusID);
	sTemp := CONCAT(sTemp, sModbusLoop);
	
	PV8 := sTemp;

//Sekvens	
	bSekvensFlagga := oaksGVL.aBModbusSekvens[iModbusLoop] = UINT_TO_INT(nUnitID);
	
	fbTempPress(
	sIPAddr:= sIpAddr, 
	nTCPPort:= INT_TO_UINT(nTCPPort), 
	nUnitID:= INT_TO_BYTE(nUnitID), 
	nQuantity:=4 , 
	nMBAddr:=0 , 
	cbLength:= SIZEOF(wArray1),
	pDestAddr:= ADR(wArray1), 
	bExecute:= bSekvensFlagga, 
	tTimeout:= T#20S, 
	bBusy=> , 
	bError=> , 
	nErrId=> , 
	cbRead=> );
	
	fbKommTof(IN:=fbTempPress.bError , PT:=T#20S , Q=> , ET=> );
	fbKommTon(IN:=fbKommTof.Q , PT:=T#20M , Q=> , ET=> );
	FAULT :=fbKommTon.Q;
	
	//Pressure
	rTemp := WORD_TO_REAL(wArray1[1]);
	PV := fSignedConverter(rInput:= rTemp);
	
	//Time constant
	PV9 := WORD_TO_UINT(wArray1[2]);
	
	//Configuration
	CASE wArray1[3] OF
	0: PV10 := '-100…100 Pa';
	1: PV10 := '0…100 Pa';
	2: PV10 := '0…200 Pa';
	3: PV10 := '0…500 Pa';
	4: PV10 := '0…1000 Pa';
	5: PV10 := '0…1500 Pa';
	6: PV10 := '0…2000 Pa';
	7: PV10 := '0…2500 Pa';
	END_CASE
	
	//Measurement output
	rTemp := WORD_TO_REAL(wArray1[4]);
	PV11 := fSignedConverter(rInput:= rTemp) / 10;
	
	//Write busy	
	oaksgvl.aBModbusBusyFlagga[iModbusLoop,nUnitID] := fbTempPress.bBusy;

END_FUNCTION_BLOCK

// oaksModbusLibrary/Produal/ProximaRIO/fbProximaCULH_RIO
//Produal Proxima CU-LH som RIO-modul. Används med givarblock för Proxima, fbProximaRIO_Sensor
//Robert H, Oaks. 24-04-08
//OBS se manual för ProximaRIO: https://oaksab.sharepoint.com/sites/Utveckling/_layouts/15/Doc.aspx?sourcedoc={22bc18e8-aa49-48c1-a1e6-a272a7cd26b5}&action=edit&wd=target%28Integrationer.one%7C5ac70296-2750-4373-ab29-5663253fae71%2FProximaRIO%20%28Produal%20Proxima%20som%20RIO%5C%29%7C3f583708-7100-47d2-8552-8b8c383d108d%2F%29&wdorigin=703
FUNCTION_BLOCK fbProximaCULH_RIO
VAR_INPUT
	
	//Allmänt
	bEnable 	: BOOL := TRUE;	//Aktivering
	bSetConfig 	: BOOL := FALSE;//Skriv konfiguration till enhet
	stModbusTCP : ST_ModbusTCP;	//Modbus-konfiguration
	nUnitID		: BYTE := 0;	//Moduladress
	tTimeOut 	: TIME := T#5S;	//Kom. timeout
		
	//IN1..3
	{attribute 'initialize_on_call'}
	rbDI1 			: REFERENCE TO BOOL;	//IN1 som digitalingång 1
	nDI1OffDelay 	: BYTE;					//Frånslagsfördröjning 0..60S (OBS opålitlig i proxima, <20s funkar dåligt och 20s blir ca 10s)
	
	{attribute 'initialize_on_call'}
	rbDI2 			: REFERENCE TO BOOL;	//IN2 som digitalingång 2
	nDI2OffDelay 	: BYTE;					//Frånslagsfördröjning 0..60S (OBS opålitlig i proxima, <20s funkar dåligt och 20s blir ca 10s)
	
	{attribute 'initialize_on_call'}
	rbDI3 			: REFERENCE TO BOOL;	//IN3 som digitalingång 3
	nDI3OffDelay 	: BYTE;					//Frånslagsfördröjning 0..60S (OBS opålitlig i proxima, <20s funkar dåligt och 20s blir ca 10s)
	
	{attribute 'initialize_on_call'}
	rfbAI1 			: REFERENCE TO fbProximaRIO_Sensor;	//IN1 som analogingång 1
	nAI1Type		: BYTE; 							//Ingångstyp (0=0..10V, 1=NTC10, 2=Ohm)
	
	{attribute 'initialize_on_call'}
	rfbAI2 			: REFERENCE TO fbProximaRIO_Sensor;	//IN2 som analogingång 2
	nAI2Type		: BYTE; 							//Ingångstyp (0=0..10V, 1=NTC10, 2=Ohm)
	
	{attribute 'initialize_on_call'}
	rfbAI3 			: REFERENCE TO fbProximaRIO_Sensor;	//IN3 som analogingång 3
	nAI3Type		: BYTE; 							//Ingångstyp (0=0..10V, 1=NTC10, 2=Ohm)
	
	//AD1 & AD2
	{attribute 'initialize_on_call'}
	rbDO1 			: REFERENCE TO BOOL;	//AD1 som digitalutgång 1
	
	{attribute 'initialize_on_call'}
	rbDO2 			: REFERENCE TO BOOL;	//AD2 som digitalutgång 2
	
	{attribute 'initialize_on_call'}
	rrAO1 			: REFERENCE TO REAL;	//AD1 som analogutgång 1 (0-10V eller PWM)
	nAO1Type		: BYTE;					//Utgångstyp (0=0-10V, 1=PWM)
	iAO1PW			: INT;					//Pulsbredd vid PWM (1..1200s)
	
	{attribute 'initialize_on_call'}
	rrAO2 : REFERENCE TO REAL;//AD2 som analogutgång 2 (0-10V eller PWM)
	nAO2Type		: BYTE;					//Utgångstyp (0=0-10V, 1=PWM)
	iAO2PW			: INT;					//Pulsbredd vid PWM (1..1200s)
	
	//AO3 & AO4
	{attribute 'initialize_on_call'}
	rrAO3 : REFERENCE TO REAL;//AO3 som analogutgång 3
	
	{attribute 'initialize_on_call'}
	rrAO4 : REFERENCE TO REAL;//AO4 som analogutgång 4
	
END_VAR
VAR_OUTPUT
	sModbusConf 	: STRING;	//Modbuskonfiguration
	bComFault 		: BOOL;		//Kommunikationsfel
	bUserFault 		: BOOL;		//Felaktigt anrop (t ex dubbel använding av ingång/utgång)
	bModuleFault	: BOOL;		//Modulfel (se sModuleFault)
	sModuleFault	: STRING;	//Orsak till modulfel
	sSerialNo		: STRING;	//Modulens serienummer (sista 8)
	bConfigOK		: BOOL;		//Konfiguration skriven
	udiComOKCnt		: UDINT := 0;	//Antal lyckade kommunikationer
	udiComErCnt		: UDINT := 0;	//Antal misslyckade kommunikationer
END_VAR
VAR
	sIP: STRING(255);
	sPort: STRING(255);
	sModbusID: STRING(255);
	sModbusLoop: STRING(255);
	sTemp : STRING(255);
	bSekvensFlagga : BOOL;
	
	aST_INConfig : ARRAY[0..2] OF ST_ProximaCULH_IO_Config;
	aST_ADConfig : ARRAY[0..3] OF ST_ProximaCULH_IO_Config;
	
	iStep: INT;
	
	nConfLoop			: BYTE := 0;
	fbMBWriteConfig		: FB_MBWriteSingleReg;
	
	nReadIOLoop			: BYTE := 0;
	fbMBReadRegs		: FB_MBReadInputRegs; 
	wInputRError		: WORD;
	wInputRSn			: WORD; 
	wInputRIo			: WORD;

	arAI_In				: ARRAY [0..2] OF REAL;
	abDI_In				: ARRAY [0..2] OF BOOL; 
	
	anADConf			: ARRAY [0..1] OF BYTE;
	arAO_Out			: ARRAY [0..3] OF REAL;
	abDO_Out			: ARRAY [0..1] OF BOOL; 
	nWriteIOLoop		: BYTE := 0;
	fbMBWriteReg		: FB_MBWriteSingleReg;
		
	//Communication error
	fbKommTof : tof; 
	fbKommTon : fbAlarm;

	R_TRIG_Sekvens: R_TRIG;
	
	bError : BOOL;
	bBusy : BOOL;
END_VAR

IF nUnitID <> 0 THEN
	
	//Övervakning sekvens	
		R_TRIG_Sekvens(CLK:= oaksGVL.aBModbusSekvens[stModbusTCP.iModbusLoop] = BYTE_TO_INT(nUnitID), Q=> bSekvensFlagga);
		
	//Sätt modbuskonfiguration på outputvariabel
		sIP := CONCAT (stModbusTCP.sIPAddr, '');
		sPort := CONCAT ('<br>Port: ', UINT_TO_STRING(stModbusTCP.nTCPPort)); 								
		sModbusID := CONCAT('<br>ID: ', BYTE_TO_STRING(nUnitID));
		sModbusLoop := CONCAT('<br>Loop: ', INT_TO_STRING(stModbusTCP.iModbusLoop));	
	
		sTemp := sIP;
		sTemp := CONCAT(sTemp, sPort);
		sTemp := CONCAT(sTemp, sModbusID);
		sTemp := CONCAT(sTemp, sModbusLoop);
		
		sModbusConf := sTemp;
	
	//Förbered konfigurationer för I/O
	
		//Kör metoder som kontrollerar hur ingångar används och sätter konfiguration
		mINConfig(rbDIChild := rbDI1, rnDIOffDelay := nDI1OffDelay, rnAIType := nAI1Type, rfbAIChild := rfbAI1, ST_Config => aST_INConfig[0]);
		mINConfig(rbDIChild := rbDI2, rnDIOffDelay := nDI2OffDelay, rnAIType := nAI2Type, rfbAIChild := rfbAI2, ST_Config => aST_INConfig[1]);
		mINConfig(rbDIChild := rbDI3, rnDIOffDelay := nDI3OffDelay, rnAIType := nAI3Type, rfbAIChild := rfbAI3, ST_Config => aST_INConfig[2]);

		//Kör metoder som kontrollerar hur utgångar används och sätter konfiguration (endast AD1/2 då AO3/4 endast är 0-10V)
		mADConfig(rbDOChild := rbDO1, rrAOChild := rrAO1, rnAOType := nAO1Type, riAOPW := iAO1PW, ST_Config => aST_ADConfig[0]);
		mADConfig(rbDOChild := rbDO2, rrAOChild := rrAO2, rnAOType := nAO2Type, riAOPW := iAO2PW, ST_Config => aST_ADConfig[1]);
		
		//Kontrollera om AO3 och AO4 används
		aST_ADConfig[2].nOutType := BOOL_TO_BYTE(__ISVALIDREF(rrAO3));	
		aST_ADConfig[3].nOutType := BOOL_TO_BYTE(__ISVALIDREF(rrAO4));
		
		//Sätt användarfel om ingångar eller utgångar används dubbelt
		bUserFault := (aST_INConfig[0].bError) OR (aST_INConfig[1].bError) OR (aST_INConfig[2].bError) OR (aST_ADConfig[0].bError) OR (aST_ADConfig[1].bError) OR (aST_ADConfig[2].bError) OR (aST_ADConfig[3].bError);
		
		
	//Modbusfunktioner i CASE-sats
		
		//Start/reset
		CASE iStep OF 
		0:
			bBusy := FALSE;
								
			IF bEnable AND bSekvensFlagga THEN
				IF bSetConfig THEN	//Gå till konfiguration om användaren önskat
					iStep := 1;
					bConfigOK := FALSE;
				ELSE				//Gå till läs/skriv I/O
					iStep := 10;
				END_IF

				bError := FALSE;
				bBusy := TRUE;
			END_IF
		
		//Konfiguration steg 1, stäng av regulator 1 & 2. Skrivning till båda genom loop
		1:	
			
			fbMBWriteConfig(
				sIPAddr:= stModbusTCP.sIPAddr, 
				nTCPPort:= stModbusTCP.nTCPPort, 
				nUnitID:= nUnitID, 
				nMBAddr:= 2100 + (nConfLoop * 100),
				nValue := 0,
				bExecute:= TRUE, 
				tTimeout:= tTimeOut);	
			
			//Gå till felsteg?
			IF fbMBWriteConfig.bError THEN fbMBWriteConfig(bExecute := FALSE); iStep := 99; END_IF
			
			//Gå vidare till nästa config-loop om OK, gå vidare till nästa steg om config-loop klar
			IF NOT fbMBWriteConfig.bBusy AND NOT fbMBWriteConfig.bError THEN 
				fbMBWriteConfig(bExecute := FALSE); 
				bError := FALSE;
				nConfLoop := nConfLoop + 1;
				
				IF nConfLoop > 1 THEN //Båda regulatorer skrivna 
					nConfLoop := 0; 
					iStep := 2; 
				END_IF;
			END_IF;
					
		
		//Konfiguration steg 2, sätt utgångar i BMS-läge (vid bSetConfig). Skrivning till samtliga genom loop			
		2:
			fbMBWriteConfig(
				sIPAddr:= stModbusTCP.sIPAddr, 
				nTCPPort:= stModbusTCP.nTCPPort, 
				nUnitID:= nUnitID, 
				nMBAddr:= 1101 + (nConfLoop * 100),
				nValue := 0,
				bExecute:= TRUE, 
				tTimeout:= tTimeOut);	
			
			//Gå till felsteg?
			IF fbMBWriteConfig.bError THEN nConfLoop := 0; fbMBWriteConfig(bExecute := FALSE); iStep := 99; END_IF
			
			//Gå vidare till nästa config-loop om OK, gå vidare till nästa steg om config-loop klar
			IF NOT fbMBWriteConfig.bBusy AND NOT fbMBWriteConfig.bError THEN 
				fbMBWriteConfig(bExecute := FALSE); 
				bError := FALSE;
				nConfLoop := nConfLoop + 1;
				
				IF nConfLoop > 3 THEN //Alla utgångar skrivna
					nConfLoop := 0; 
					iStep := 3; 
				END_IF;
			END_IF; 

		//Konfiguration steg 3, sätt utgångar i överstyrningsläge (vid bSetConfig). Skrivning till samtliga genom loop		
		3:
			fbMBWriteConfig(
				sIPAddr:= stModbusTCP.sIPAddr, 
				nTCPPort:= stModbusTCP.nTCPPort, 
				nUnitID:= nUnitID, 
				nMBAddr:= 1113 + (nConfLoop * 100),
				nValue := 1,
				bExecute:= TRUE, 
				tTimeout:= tTimeOut);	
			
			//Gå till felsteg?
			IF fbMBWriteConfig.bError THEN nConfLoop := 0; fbMBWriteConfig(bExecute := FALSE); iStep := 99; END_IF
			
			//Gå vidare till nästa config-loop om OK, gå vidare till nästa steg om config-loop klar
			IF NOT fbMBWriteConfig.bBusy AND NOT fbMBWriteConfig.bError THEN 
				fbMBWriteConfig(bExecute := FALSE); 
				bError := FALSE;
				nConfLoop := nConfLoop + 1;
				
				IF nConfLoop > 3 THEN //Alla utgångar skrivna 
					nConfLoop := 0; 
					iStep := 4; 
				END_IF;
			END_IF; 		
		
		//Konfiguration steg 4, sätt snabb reaktionstid på alla ingångar. Skrivning till samtliga genom loop
		4:
			fbMBWriteConfig(
				sIPAddr:= stModbusTCP.sIPAddr, 
				nTCPPort:= stModbusTCP.nTCPPort, 
				nUnitID:= nUnitID, 
				nMBAddr:= 135 + (nConfLoop * 100),
				nValue := 1,
				bExecute:= TRUE, 
				tTimeout:= tTimeOut);	
			
			//Gå till felsteg?
			IF fbMBWriteConfig.bError THEN nConfLoop := 0; fbMBWriteConfig(bExecute := FALSE); iStep := 99; END_IF
			
			//Gå vidare till nästa config-loop om OK, gå vidare till nästa steg om config-loop klar
			IF NOT fbMBWriteConfig.bBusy AND NOT fbMBWriteConfig.bError THEN 
				fbMBWriteConfig(bExecute := FALSE); 
				bError := FALSE;
				nConfLoop := nConfLoop + 1;
				
				IF nConfLoop > 2 THEN //Alla ingångar skrivna 
					nConfLoop := 0; 
					iStep := 5; 
				END_IF;
			END_IF;

		//Konfiguration steg 5, sätt ingångstyper. Skrivning till samtliga genom loop
		5: 	
			fbMBWriteConfig(
				sIPAddr:= stModbusTCP.sIPAddr, 
				nTCPPort:= stModbusTCP.nTCPPort, 
				nUnitID:= nUnitID, 
				nMBAddr:= 100 + (nConfLoop * 100),
				nValue := aST_INConfig[nConfLoop].nInType,
				bExecute:= TRUE, 
				tTimeout:= tTimeOut);	
				
			//Gå till felsteg?
			IF fbMBWriteConfig.bError THEN nConfLoop := 0; fbMBWriteConfig(bExecute := FALSE); iStep := 99; END_IF
			
			//Gå vidare till nästa config-loop om OK, gå vidare till nästa steg om config-loop klar
			IF NOT fbMBWriteConfig.bBusy AND NOT fbMBWriteConfig.bError THEN 
				fbMBWriteConfig(bExecute := FALSE); 
				bError := FALSE;
				nConfLoop := nConfLoop + 1;
				
				IF nConfLoop > 2 THEN //Alla ingångar skrivna 
					nConfLoop := 0; 
					iStep := 6; 
				END_IF;
			END_IF; 
		
		//Konfiguration steg 6, sätt fördröjning för konfigurerade digitalingångar. Skrivning till samtliga genom loop
		6: 	
			fbMBWriteConfig(
				sIPAddr:= stModbusTCP.sIPAddr, 
				nTCPPort:= stModbusTCP.nTCPPort, 
				nUnitID:= nUnitID, 
				nMBAddr:= 121 + (nConfLoop * 100),	//Skriv till ondelay då DI är inverterad
				nValue := aST_INConfig[nConfLoop].nInDelay,
				bExecute:= (aST_INConfig[nConfLoop].nInType = 7) AND (aST_INConfig[nConfLoop].nInDelay > 0), 
				tTimeout:= tTimeOut);	
				
			//Gå till felsteg?
			IF fbMBWriteConfig.bError THEN nConfLoop := 0; fbMBWriteConfig(bExecute := FALSE); iStep := 99; END_IF
			
			//Gå vidare till nästa config-loop om OK, gå vidare till nästa steg om config-loop klar
			IF NOT fbMBWriteConfig.bBusy AND NOT fbMBWriteConfig.bError THEN 
				fbMBWriteConfig(bExecute := FALSE); 
				bError := FALSE;
				nConfLoop := nConfLoop + 1;
				
				IF nConfLoop > 2 THEN //Alla ingångar skrivna 
					nConfLoop := 0; 
					iStep := 7; 
				END_IF;
			END_IF; 
			
		//Konfiguration steg 7, sätt utgångstyper. Skrivning till samtliga genom loop
		7: 	
			fbMBWriteConfig(
				sIPAddr:= stModbusTCP.sIPAddr, 
				nTCPPort:= stModbusTCP.nTCPPort, 
				nUnitID:= nUnitID, 
				nMBAddr:= 1100 + (nConfLoop * 100),
				nValue := aST_ADConfig[nConfLoop].nOutType,
				bExecute:= TRUE, 
				tTimeout:= tTimeOut);	
				
			//Gå till felsteg?
			IF fbMBWriteConfig.bError THEN nConfLoop := 0; fbMBWriteConfig(bExecute := FALSE); iStep := 99; END_IF
			
			//Gå vidare till nästa config-loop om OK, gå vidare till nästa steg om config-loop klar
			IF NOT fbMBWriteConfig.bBusy AND NOT fbMBWriteConfig.bError THEN 
				fbMBWriteConfig(bExecute := FALSE); 
				bError := FALSE;
				nConfLoop := nConfLoop + 1;
				
				IF nConfLoop > 3 THEN //Alla utgångar skrivna 
					nConfLoop := 0; 
					iStep := 8; 
				END_IF;
			END_IF;

		//Konfiguration steg 8, sätt pulstid för AD-utgångar. Skrivning till samtliga genom loop
		8: 	
			fbMBWriteConfig(
				sIPAddr:= stModbusTCP.sIPAddr, 
				nTCPPort:= stModbusTCP.nTCPPort, 
				nUnitID:= nUnitID, 
				nMBAddr:= 1138 + (nConfLoop * 100),
				nValue := aST_ADConfig[nConfLoop].iOutPW,
				bExecute:= TRUE, 
				tTimeout:= tTimeOut);	
			
			//Gå till felsteg?
			IF fbMBWriteConfig.bError THEN nConfLoop := 0; fbMBWriteConfig(bExecute := FALSE); iStep := 99; END_IF
			
			//Gå vidare till nästa config-loop om OK, om config-loop klar sätt bConfigOK och gå till steg 10 (läs/skriv I/O)
			IF NOT fbMBWriteConfig.bBusy AND NOT fbMBWriteConfig.bError THEN 
				fbMBWriteConfig(bExecute := FALSE); 
				bError := FALSE;
				nConfLoop := nConfLoop + 1;
				
				IF nConfLoop > 1 THEN //Alla utgångar skrivna
					bConfigOK := TRUE;
					bSetConfig := FALSE;
					nConfLoop := 0; 
					iStep := 10; 
				END_IF;
			END_IF; 
		
		//Läs felregister
		10:
			fbMBReadRegs(
				sIPAddr:= stModbusTCP.sIpAddr, 
				nTCPPort:= stModbusTCP.nTCPPort, 
				nUnitID:= nUnitID, 
				nQuantity:= 1,
				nMBAddr:= 0, 
				cbLength:= SIZEOF(wInputRError), 
				pDestAddr:= ADR(wInputRError), 
				bExecute:= TRUE, 
				tTimeout:= tTimeOut);
				
			//Gå till felsteg?
			IF fbMBReadRegs.bError THEN fbMBReadRegs(bExecute := FALSE); iStep := 99; END_IF

			//Överför värden och gå vidare till nästa steg om OK
			IF NOT fbMBReadRegs.bBusy AND NOT fbMBReadRegs.bError THEN
				
				bModuleFault := wInputRError.0 OR wInputRError.3;
				IF wInputRError.0 THEN sModuleFault := 'Låg spänning'; END_IF
				IF wInputRError.3 THEN sModuleFault := 'Fel programvaruversion'; END_IF
				IF NOT bModuleFault THEN sModuleFault := 'Inget fel'; END_IF
				
				fbMBReadRegs(bExecute := FALSE); 
				bError := FALSE;
				iStep := 11;
			END_IF;
			
		//Läs serienummer
		11:
			fbMBReadRegs(
				sIPAddr:= stModbusTCP.sIpAddr, 
				nTCPPort:= stModbusTCP.nTCPPort, 
				nUnitID:= nUnitID, 
				nQuantity:= 1,
				nMBAddr:= 9903, 
				cbLength:= SIZEOF(wInputRSn), 
				pDestAddr:= ADR(wInputRSn), 
				bExecute:= TRUE, 
				tTimeout:= tTimeOut);
				
			//Gå till felsteg?
			IF fbMBReadRegs.bError THEN fbMBReadRegs(bExecute := FALSE); iStep := 99; END_IF

			//Överför värden och gå vidare till nästa steg om OK
			IF NOT fbMBReadRegs.bBusy AND NOT fbMBReadRegs.bError THEN
				
				sSerialNo := WORD_TO_HEXSTR(in := wInputRSn, iPrecision := 8, bLoCase := FALSE);
				
				fbMBReadRegs(bExecute := FALSE); 
				bError := FALSE;
				iStep := 12;
			END_IF;
			
		//Läs ingångar. Läsning av samtliga genom loop (läser ej avstängda eller felkonfigurerade ingångar). Samt justering av register som läses enligt typ
		12:
			IF aST_INConfig[nReadIOLoop].nInType <> 0 THEN
				
				IF aST_INConfig[nReadIOLoop].nInType = 1 THEN		//0-10V
					 fbMBReadRegs.nMBAddr := 101;
				ELSIF aST_INConfig[nReadIOLoop].nInType = 5 THEN	//NTC
					fbMBReadRegs.nMBAddr := 104;
				ELSIF aST_INConfig[nReadIOLoop].nInType = 7 THEN	//Res
					IF aST_INConfig[nReadIOLoop].nInRType = 0 THEN	//Ohm
						fbMBReadRegs.nMBAddr := 102;
					ELSE											//DI
						fbMBReadRegs.nMBAddr := 107;
					END_IF
				END_IF;
				
				fbMBReadRegs.nMBAddr := fbMBReadRegs.nMBAddr + (nReadIOLoop * 100);
			
				fbMBReadRegs(
					sIPAddr:= stModbusTCP.sIpAddr, 
					nTCPPort:= stModbusTCP.nTCPPort, 
					nUnitID:= nUnitID, 
					nQuantity:= 1,
					cbLength:= SIZEOF(wInputRIo), 
					pDestAddr:= ADR(wInputRIo), 
					bExecute:= TRUE, 
					tTimeout:= tTimeOut);
				
				//Gå till felsteg?
				IF fbMBReadRegs.bError THEN fbMBReadRegs(bExecute := FALSE); iStep := 99; END_IF
	
				//Överför värden och gå vidare till nästa läsloopom OK, gå vidare till nästa steg om läsloopom klar. Överför till rätt outputs beroende på IO-typ
				IF NOT fbMBReadRegs.bBusy AND NOT fbMBReadRegs.bError THEN
					
					IF aST_INConfig[nReadIOLoop].nInType = 1 THEN		//0-10V, omvandla till råvärde 0-10V (skalning görs i givarblock)
						arAI_In[nReadIOLoop] := INT_TO_REAL(WORD_TO_INT(wInputRIo)) / 1000; 
					ELSIF aST_INConfig[nReadIOLoop].nInType = 5 THEN	//NTC, omvlandla till temperatur med en decimal
						arAI_In[nReadIOLoop] := INT_TO_REAL(WORD_TO_INT(wInputRIo)) / 10; 
					ELSIF aST_INConfig[nReadIOLoop].nInType = 7 THEN	//Res
						IF aST_INConfig[nReadIOLoop].nInRType = 0 THEN	//Ohm, omvandla till ohm x 10
							arAI_In[nReadIOLoop] := INT_TO_REAL(WORD_TO_INT(wInputRIo)) * 10; 
						ELSE											//DI, läs bit 0 inverterat
							abDI_In[nReadIOLoop] := NOT wInputRIo.0;
						END_IF
					END_IF;
					
					fbMBReadRegs(bExecute := FALSE); 
					bError := FALSE;
					nReadIOLoop := nReadIOLoop + 1;
					
					IF nReadIOLoop > 2 THEN //Alla ingångar lästa 
						nReadIOLoop := 0; 
						iStep := 13; 
					END_IF;
				
				END_IF
			
			ELSE	//Ej använd eller felkonfigurerad ingång
				nReadIOLoop := nReadIOLoop + 1;
				
				IF nReadIOLoop > 2 THEN //Alla ingångar lästa 
					nReadIOLoop := 0; 
					iStep := 13; 
				END_IF;
			END_IF;
			
			//Skriv ingångsvärden till anslutna variabler
			IF __ISVALIDREF(rbDI1) THEN rbDI1 := abDI_In[0]; END_IF;
			IF __ISVALIDREF(rbDI2) THEN rbDI2 := abDI_In[1]; END_IF;
			IF __ISVALIDREF(rbDI3) THEN rbDI3 := abDI_In[2]; END_IF;
			
			IF __ISVALIDREF(rfbAI1) THEN rfbAI1.mDataIn(rInVal := arAI_In[0], nInType := nAI1Type); END_IF;
			IF __ISVALIDREF(rfbAI2) THEN rfbAI2.mDataIn(rInVal := arAI_In[1], nInType := nAI2Type); END_IF;
			IF __ISVALIDREF(rfbAI3) THEN rfbAI3.mDataIn(rInVal := arAI_In[2], nInType := nAI3Type); END_IF;
		
		//Skriv utgångar. Skrivning av samtliga genom loop (skriver ej avstängda eller felkonfigurerade utgångar). Samt justering av värde som skrivs enligt typ	
		13:
			//Skriv AD1/2 utgångstyper till array för AD1/2
			anADConf[0] := nAO1Type;
			anADConf[1] := nAO2Type;
			
			//Skriv referensvärden till array för analoga ut
			IF __ISVALIDREF(rrAO1) THEN arAO_Out[0] := rrAO1; END_IF;
			IF __ISVALIDREF(rrAO2) THEN arAO_Out[1] := rrAO2; END_IF;
			IF __ISVALIDREF(rrAO3) THEN arAO_Out[2] := rrAO3; END_IF;
			IF __ISVALIDREF(rrAO4) THEN arAO_Out[3] := rrAO4; END_IF;
			
			//Skriv referensvärden till array för digitala ut
			IF __ISVALIDREF(rbDO1) THEN abDO_Out[0] := rbDO1; END_IF;
			IF __ISVALIDREF(rbDO2) THEN abDO_Out[1] := rbDO2; END_IF;  
			
			
			IF aST_ADConfig[nWriteIOLoop].nOutType <> 0 THEN
				
				IF aST_ADConfig[nWriteIOLoop].nOutType = 1 THEN		//0-100% -> 0-10000
					 fbMBWriteReg.nValue := REAL_TO_WORD(arAO_Out[nWriteIOLoop] * 100);
				ELSIF (aST_ADConfig[nWriteIOLoop].nOutType = 4) AND (nWriteIOLoop <= 1) THEN	//DO / PWM
					IF anADConf[nWriteIOLoop] = 0 THEN				//DO -> 0 / 10000
						fbMBWriteReg.nValue := 10000 * BOOL_TO_WORD(abDO_Out[nWriteIOLoop]);
					ELSE											//PWM -> 0-100% - 0-10000
						fbMBWriteReg.nValue := REAL_TO_WORD(arAO_Out[nWriteIOLoop] * 100);
					END_IF
						
				END_IF;
			
				fbMBWriteReg(
					sIPAddr:= stModbusTCP.sIPAddr, 
					nTCPPort:= stModbusTCP.nTCPPort, 
					nUnitID:= nUnitID, 
					nMBAddr:= 1114 + (nWriteIOLoop * 100),
					bExecute:= TRUE, 
					tTimeout:= tTimeOut);	
				
				//Gå till felsteg?
				IF fbMBWriteReg.bError THEN fbMBWriteReg(bExecute := FALSE); iStep := 99; END_IF
	
				//Överför värden och gå vidare till nästa läsloopom OK, gå vidare till nästa steg om läsloopom klar. Överför till rätt outputs beroende på IO-typ
				IF NOT fbMBWriteReg.bBusy AND NOT fbMBWriteReg.bError THEN
					
					fbMBWriteReg(bExecute := FALSE); 
					bError := FALSE;
					nWriteIOLoop := nWriteIOLoop + 1;
					
					IF nWriteIOLoop > 3 THEN //Alla utgångar skrivna 
						nWriteIOLoop := 0; 
						iStep := 20; 
					END_IF;
				
				END_IF
			
			ELSE	//Ej använd eller felkonfigurerad ingång
				nWriteIOLoop := nWriteIOLoop + 1;
				
				IF nWriteIOLoop > 3 THEN //Alla utgångar skrivna 
					nWriteIOLoop := 0; 
					iStep := 20; 
				END_IF;
			END_IF;

		//Succe			
		20:
			udiComOKCnt := udiComOKCnt + 1;
			bBusy := FALSE;
			iStep := 0;
			
		//Felhantering
		99:
			udiComErCnt := udiComErCnt + 1;
			bBusy := FALSE;
			bError := TRUE;
			iStep := 0;

		END_CASE;
		
END_IF;

//Kommunikationsfel modul
	fbKommTof(IN:=bError , PT:=T#20S , Q=> , ET=> );
	fbKommTon(bInput:=fbKommTof.Q , tAlarmDelay:=T#1M , bAutoReset:= , bAlarmOutput=> );
	bComFault := fbKommTon.bAlarmOutput OR (nUnitID = 0);
			
//Rapportera upptagen enhet	
	oaksgvl.aBModbusBusyFlagga[stModbusTCP.iModbusLoop,nUnitID] := bBusy;

//Sätter unika konfiguration för AD-utgångar
METHOD PRIVATE mADConfig

VAR_INPUT
	rbDOChild		: REFERENCE TO BOOL;
	rrAOChild		: REFERENCE TO REAL;
	rnAOType		: REFERENCE TO BYTE;
    riAOPW			: REFERENCE TO INT;	
END_VAR

VAR_OUTPUT
	ST_Config	: ST_ProximaCULH_IO_Config;
END_VAR
//Kontrollera hur ingången används
ST_Config.bError := FALSE;

IF __ISVALIDREF(rbDOChild) AND __ISVALIDREF(rrAOChild) THEN	//Båda (fel) 
	ST_Config.nInType := 0;
	ST_Config.bError := TRUE;
	
ELSIF __ISVALIDREF(rrAOChild) THEN //AO/PWM
	IF rnAOType = 0 THEN
		ST_Config.nOutType := 1;
	ELSIF rnAOType = 1 THEN
		ST_Config.nOutType := 4;
		ST_Config.iOutPW := riAOPW; 
	END_IF;
	
ELSIF __ISVALIDREF(rbDOChild) THEN //DO
	ST_Config.nOutType := 4;
	ST_Config.iOutPW := 1;

ELSE //Ingen, används ej
	ST_Config.nOutType := 0;
END_IF
END_METHOD

//Sätter unika konfiguration för ingångar
METHOD PRIVATE mINConfig

VAR_INPUT
	rbDIChild		: REFERENCE TO BOOL;
	rnDIOffDelay 	: REFERENCE TO BYTE;
	rfbAIChild		: REFERENCE TO fbProximaRIO_Sensor;
	rnAIType		: REFERENCE TO BYTE;	
END_VAR

VAR_OUTPUT
	ST_Config	: ST_ProximaCULH_IO_Config;
END_VAR
//Kontrollera hur ingången används
ST_Config.bError := FALSE;

IF __ISVALIDREF(rbDIChild) AND __ISVALIDREF(rfbAIChild) THEN	//Båda (fel) 
	ST_Config.nInType := 0;
	ST_Config.bError := TRUE;
	
ELSIF __ISVALIDREF(rfbAIChild) THEN //AI
	IF rnAIType = 0 THEN
		ST_Config.nInType := 1;
	ELSIF rnAIType = 1 THEN
		ST_Config.nInType := 5;
	ELSIF rnAIType = 2 THEN
		ST_Config.nInType := 7;
		ST_Config.nInRType := 0;
	END_IF;
	
ELSIF __ISVALIDREF(rbDIChild) THEN //DI
	ST_Config.nInType := 7;
	ST_Config.nInRType := 1;
	ST_Config.nInDelay := rnDIOffDelay;

ELSE //Ingen, används ej
	ST_Config.nInType := 0;
END_IF
END_METHOD

END_FUNCTION_BLOCK

// oaksModbusLibrary/Produal/ProximaRIO/fbProximaRIO_Sensor
//Givarblock för Proxima CU-LH som RIO (används med fbProximaCULH_RIO)
//OBS se manual för ProximaRIO: https://oaksab.sharepoint.com/sites/Utveckling/_layouts/15/Doc.aspx?sourcedoc={22bc18e8-aa49-48c1-a1e6-a272a7cd26b5}&action=edit&wd=target%28Integrationer.one%7C5ac70296-2750-4373-ab29-5663253fae71%2FProximaRIO%20%28Produal%20Proxima%20som%20RIO%5C%29%7C3f583708-7100-47d2-8552-8b8c383d108d%2F%29&wdorigin=703
FUNCTION_BLOCK fbProximaRIO_Sensor
VAR_INPUT
	rAISclRawMin	: REAL := 0;		//Min skalning råvärde för aktiv givare (0..10V) 
	rAISclRawMax	: REAL := 10;		//Max skalning råvärde för aktiv givare (0..10V)
	rAISclEngMin	: REAL := 0;		//Min skalning för aktiv givare i ingenjörsenhet
	rAISclEngMax	: REAL := 100;		//Max skalning för aktiv givare i ingenjörsenhet
	udiDamp			: UDINT := 0;		//Dämpning av givarvärde (sekunder)
	bUseFault		: BOOL := TRUE;		//Givarfel på/av (0..10V / Ohm = givarfel om råvärde under/över min/max, NTC = Givarfel om värde <=40 eller >=140 
	tAlarmDelay		: TIME := T#1S;		//Larmfördröjning givarfel
END_VAR

VAR_OUTPUT
	rPV 			: REAL;		//Givarvärde 
	bFAULT		 	: BOOL;		//Givarfel
END_VAR

VAR
	rInVal 	: REAL;
	nInType	: BYTE;
	bFaultInt	: BOOL;
	rPVint		: REAL;
	fbDamp	: Tc3_BA.FB_BA_TiAvrg;
	fbFault	: fbAlarm;											
END_VAR

IF nInType = 0 THEN			//0-10V
	bFaultInt := (rInVal < rAISclRawMin) OR (rInVal > rAISclRawMax);	//Givarfel om råvärde utanför angivet område
	rPVint := fScale2p(rX := rInVal, X1 := rAISclRawMin, X2 := rAISclRawMax, Y1 := rAISclEngMin, Y2 := rAISclEngMax);	//Beräkna PV linjärt enligt råvärde & ing.enhet min/max
ELSIF nInType = 1 THEN		//NTC10
	bFaultInt := (rInVal <= -40) OR (rInVal > 140);					//Givarfel om orimligt lågt/högt värde
	rPVint	:= rInVal;
ELSIF nInType = 2 THEN		//Ohm
	bFaultInt := (rInVal < rAISclRawMin) OR (rInVal > rAISclRawMax);	//Givarfel om råvärde utanför angivet område
	rPVint := rInVal;
END_IF

IF udiDamp > 0 THEN	//Dämpa givarvärde eller skriv det utan dämpning
	fbDamp(bEn := TRUE, rIn := rPVint, udiIntval_sec := 1, udiNumOfElem := udiDamp, rOut => rPV);
ELSE
	rPV := rPVint;
END_IF

fbFault(bInput := bFaultInt AND bUseFault, tAlarmDelay := tAlarmDelay, bAutoReset := TRUE, bAlarmOutput => bFAULT);	//Givarfelslarm

METHOD PUBLIC mDataIn : REAL
VAR_INPUT
	rInVal : REAL;
	nInType : BYTE;
END_VAR
THIS^.rInVal := rInVal;
THIS^.nInType := nInType;
END_METHOD

END_FUNCTION_BLOCK

// oaksModbusLibrary/Produal/Regulatorer/HLS44/fbProdualHLS44
//Oaks AB
//2022-08-19
//Funktionsblock för styrning av Produal HLS44
FUNCTION_BLOCK fbProdualHLS44
VAR_INPUT
	sIPAddr : STRING := '127.0.0.1'; 
	nTCPPort : UINT := 502;
	nUnitID : UINT :=1;
	iModbusLoop : INT :=1; //Modbusslinga
	tTimeout : TIME := T#3S; //Timeout
	bResetUserSetpoint : BOOL; //Återställ lokal förskjutning
	bNightMode : BOOL := FALSE; //Aktivera nattläge
		
	bCoolOutputA1override : BOOL :=FALSE; //Överstyr kylutgång
	rCoolOutputA1override : REAL :=0; //Kylutgång (0-100%)
	
	bHeatOutputA2override : BOOL := FALSE; //Överstyr värmeutgång
	rHeatOutputA2override : REAL :=0; //Värmeutgång (0-100%)
	bVavOutputY1override : BOOL := FALSE; //Överstyr VAV-utgång
	rVavOutputY1override : REAL :=0; //VAV-utgång (0-100%)
	
END_VAR

VAR_OUTPUT
	{attribute 'OPC.UA.DA' := '1'}
	PV AT %M* : REAL;//Temperatur~wp:[unit]°C[format]0.0
	{attribute 'OPC.UA.DA' := '1'}
	PV1 AT %M* : REAL;//Koldioxidhalt~wp:[unit]ppm[format]0
	{attribute 'OPC.UA.DA' := '1'}
	CSP AT %M* : REAL;//Uträknat börvärde~wp:[unit]°C[format]0.0
	{attribute 'OPC.UA.DA' := '1'}
	PV2 AT %M* : REAL;//Förskjutning börvärde från användare~wp:[unit]°C[format]0.0
	{attribute 'OPC.UA.DA' := '1'}
	PV8 AT %M* : STRING;//Modbus konfiguering~wp:
	{attribute 'OPC.UA.DA' := '1'}
	FAULT AT %M* : BOOL;//Kommunikationsfel~wp:
	
	rCoolOutputA1 : REAL :=0; //Kylutgång	(0-100%)
	rHeatOutputA2 : REAL :=0; //Värmeutgång (0-100%)
	rVavOutputY1 : REAL :=0; //VAV-utgång (0-100%)
END_VAR

VAR
	bSekvensFlagga : BOOL;
			
	FB_MBReadRegs_InputRegs1: FB_MBReadInputRegs;
	ArrHolding1 : ARRAY [0..21] OF WORD; //Holding
		
	//Kommunikationsfel
	fbKommTof : tof; 
	fbKommTon : fbAlarm;
	
	sIP: STRING(255);
	sPort: STRING(255);
	sModbusID: STRING(255);
	sModbusLoop: STRING(255);
	sTemp : STRING(255);
	
	fbReadWriteHoldingRegReal_Sp: fbReadWriteHoldingRegReal;
	F_TRIG_Steg1: F_TRIG;
	F_TRIG_Steg2: F_TRIG;
	F_TRIG_Steg3: F_TRIG;
	F_TRIG_Steg4: F_TRIG;
	F_TRIG_Steg5: F_TRIG;
	F_TRIG_Steg6: F_TRIG;
	F_TRIG_Steg7: F_TRIG;
	F_TRIG_Steg8: F_TRIG;
	F_TRIG_Steg9: F_TRIG;
	fbReadWriteHoldingRegReal_Offset: fbReadWriteHoldingRegReal;
	rOffsetToWrite: REAL;
	fbReadWriteCoilRegBool_Night: fbReadWriteCoilRegBool;
	fbReadWriteCoilRegBool_A1: fbReadWriteCoilRegBool;
	fbReadWriteHoldingRegReal_A1: fbReadWriteHoldingRegReal;
	fbReadWriteCoilRegBool_A2: fbReadWriteCoilRegBool;
	fbReadWriteHoldingRegReal_A2: fbReadWriteHoldingRegReal;
	fbReadWriteCoilRegBool_Y1: fbReadWriteCoilRegBool;
	fbReadWriteHoldingRegReal_Y1: fbReadWriteHoldingRegReal;
	rSetpointToWrite : REAL;
	wWordToWrite: WORD;
	F_TRIG_Steg10: F_TRIG;
	fbReadWriteHoldingRegReal_Setpoint: fbReadWriteHoldingRegReal;
	R_TRIG_start: R_TRIG;
	bBusy: BOOL;
END_VAR

VAR_INPUT PERSISTENT
	{attribute 'OPC.UA.DA' := '1'}
	SP1 AT %M* : REAL := 21;//Rumsbörvärde~wp:[unit]°C[format]0.0
	{attribute 'OPC.UA.DA' := '1'}
	SP3 AT %M* : REAL := 0;//Max förskjutning börvärde +/-~wp:[unit]°C[format]0.0
	{attribute 'OPC.UA.DA' := '1'}
	SP4 AT %M* : REAL := 0;//Justering av temperaturgivare~wp:[unit]°C[format]0.0
END_VAR

//Sekvens	
	bSekvensFlagga := oaksGVL.aBModbusSekvens[iModbusLoop] = UINT_TO_INT(nUnitID);
//Modbus konfiguering
	sIP := CONCAT (SIPAddr, '');
	sPort := CONCAT ('<br>Port: ', UINT_TO_STRING(nTCPPort)); 								
	sModbusID := CONCAT('<br>ID: ', UINT_TO_STRING(nUnitID));
	sModbusLoop := CONCAT('<br>Loop: ', INT_TO_STRING(iModbusLoop));	

	sTemp := sIP;
	sTemp := CONCAT(sTemp, sPort);
	sTemp := CONCAT(sTemp, sModbusID);
	sTemp := CONCAT(sTemp, sModbusLoop);
	
	PV8 := sTemp;

///////////////		
//READ
///////////////		

	R_TRIG_start(CLK:= bSekvensFlagga, Q=> );
		
	//Read Holding 0-10
	FB_MBReadRegs_InputRegs1(
	sIPAddr:= sIpAddr, 
	nTCPPort:= INT_TO_UINT(nTCPPort), 
	nUnitID:= INT_TO_BYTE(nUnitID), 
	nQuantity:= 22, 
	nMBAddr:= 0 , 
	cbLength:= SIZEOF(ArrHolding1), 
	pDestAddr:= ADR(ArrHolding1), 
	bExecute:= R_TRIG_start.Q, 
	tTimeout:= tTimeout, 
	bBusy=> , 
	bError=> , 
	nErrId=> , 
	cbRead=> );
	
		//Values
		//ArrHolding1[0]; //0
		//ArrHolding1[1]; //1
		//ArrHolding1[2]; //2
		PV := fSignedConverter(WORD_TO_REAL(ArrHolding1[3])) /10; //4
		//ArrHolding1[4]; //4
		PV1 := fSignedConverter(WORD_TO_REAL(ArrHolding1[5])); //5
		CSP := fSignedConverter(WORD_TO_REAL(ArrHolding1[6])) /10; //6
		//rCoolOutputA1 := fSignedConverter(WORD_TO_REAL(ArrHolding1[7]) / 10); //7 delat med 10 för att slippa konvertera från 0-10V -> 0-100%
		//rHeatOutputA2 := fSignedConverter(WORD_TO_REAL(100-(ArrHolding1[8]) /10)); //8 delat med 10 för att slippa konvertera från 0-10V -> 0-100%
		//ArrHolding1[9]; //9
		//ArrHolding1[10]; //10
		rVavOutputY1 := fSignedConverter(WORD_TO_REAL(ArrHolding1[11])) /10; //11 delat med 10 för att slippa konvertera från 0-10V -> 0-100%
		//ArrHolding1[12]; //12
		//ArrHolding1[13]; //13
		//ArrHolding1[14]; //14
		//ArrHolding1[15]; //15
		//ArrHolding1[16]; //16
		//ArrHolding1[17]; //17
		//ArrHolding1[18]; //18
		
		PV2 := fSignedConverter(WORD_TO_REAL(ArrHolding1[19])) /10;
		rCoolOutputA1 := fSignedConverter(WORD_TO_REAL(ArrHolding1[20])) /10; //7 delat med 10 för att slippa konvertera från 0-10V -> 0-100%
		rHeatOutputA2 := 100 - fSignedConverter(WORD_TO_REAL((ArrHolding1[21])) /10); //8 delat med 10 för att slippa konvertera från 0-10V -> 0-100%
		
///////////////		
//WRITE
///////////////			

//Write centre of user setpoint area

rSetpointToWrite := SP1;

F_TRIG_Steg1(CLK:= FB_MBReadRegs_InputRegs1.bBusy, Q=> );

fbReadWriteHoldingRegReal_Sp(
	sIPAddr:= sIpAddr, 
	nTCPPort:= INT_TO_UINT(nTCPPort), 
	nUnitID:= INT_TO_BYTE(nUnitID), 
	mBusAdr:= 10, 
	bEnable:= F_TRIG_Steg1.Q, 
	tTimeout:= tTimeout, 
	rReal:= rSetpointToWrite, 
	uiFaktor:= 10, 
	bError=> , 
	bBusy=> , 
	bSuccess=> );

//Write centre of user setpoint area	
IF bResetUserSetpoint THEN
	rOffsetToWrite := 0;
ELSE
	rOffsetToWrite := SP3;
END_IF

F_TRIG_Steg2(CLK:= fbReadWriteHoldingRegReal_Sp.bBusy, Q=> );

fbReadWriteHoldingRegReal_Offset(
	sIPAddr:= sIpAddr, 
	nTCPPort:= INT_TO_UINT(nTCPPort), 
	nUnitID:= INT_TO_BYTE(nUnitID), 
	mBusAdr:= 11, 
	bEnable:= F_TRIG_Steg2.Q, 
	tTimeout:= tTimeout, 
	rReal:= rOffsetToWrite, 
	uiFaktor:= 10, 
	bError=> , 
	bBusy=> , 
	bSuccess=> );

F_TRIG_Steg3(CLK:= fbReadWriteHoldingRegReal_Offset.bBusy, Q=> );
	
	fbReadWriteCoilRegBool_Night(
	sIPAddr:= sIpAddr, 
	nTCPPort:= INT_TO_UINT(nTCPPort), 
	nUnitID:= INT_TO_BYTE(nUnitID), 
	mBusAdr:= 13, 
	bEnable:= F_TRIG_Steg3.Q, 
	tTimeout:= tTimeout, 
	bBool:= bNightMode, 
	bError=> , 
	bBusy=> , 
	bSuccess=> );

//Override A1
F_TRIG_Steg4(CLK:= fbReadWriteCoilRegBool_Night.bBusy, Q=> );
	
	fbReadWriteCoilRegBool_A1(
	sIPAddr:= sIpAddr, 
	nTCPPort:= INT_TO_UINT(nTCPPort), 
	nUnitID:= INT_TO_BYTE(nUnitID), 
	mBusAdr:= 0, 
	bEnable:= F_TRIG_Steg4.Q, 
	tTimeout:= tTimeout, 
	bBool:= bCoolOutputA1override, 
	bError=> , 
	bBusy=> , 
	bSuccess=> );
	
F_TRIG_Steg5(CLK:= fbReadWriteCoilRegBool_A1.bBusy, Q=> );
	
	fbReadWriteHoldingRegReal_A1(
	sIPAddr:= sIpAddr, 
	nTCPPort:= INT_TO_UINT(nTCPPort), 
	nUnitID:= INT_TO_BYTE(nUnitID), 
	mBusAdr:= 2, 
	bEnable:= F_TRIG_Steg5.Q, 
	tTimeout:= tTimeout, 
	rReal:= LIMIT(0,rCoolOutputA1override,100), 
	uiFaktor:= 10, 
	bError=> , 
	bBusy=> , 
	bSuccess=> );
	
//Override A2
F_TRIG_Steg6(CLK:= fbReadWriteHoldingRegReal_A1.bBusy, Q=> );
	
	fbReadWriteCoilRegBool_A2(
	sIPAddr:= sIpAddr, 
	nTCPPort:= INT_TO_UINT(nTCPPort), 
	nUnitID:= INT_TO_BYTE(nUnitID), 
	mBusAdr:= 2, 
	bEnable:= F_TRIG_Steg6.Q, 
	tTimeout:= tTimeout, 
	bBool:= bHeatOutputA2override, 
	bError=> , 
	bBusy=> , 
	bSuccess=> );
	
F_TRIG_Steg7(CLK:= fbReadWriteCoilRegBool_A2.bBusy, Q=> );
	
	fbReadWriteHoldingRegReal_A2(
	sIPAddr:= sIpAddr, 
	nTCPPort:= INT_TO_UINT(nTCPPort), 
	nUnitID:= INT_TO_BYTE(nUnitID), 
	mBusAdr:= 4, 
	bEnable:= F_TRIG_Steg7.Q, 
	tTimeout:= tTimeout, 
	rReal:= LIMIT(0,(100-rHeatOutputA2override),100), 
	uiFaktor:= 10, 
	bError=> , 
	bBusy=> , 
	bSuccess=> );	

//Override Y1
F_TRIG_Steg8(CLK:= fbReadWriteHoldingRegReal_A2.bBusy, Q=> );
	
	fbReadWriteCoilRegBool_Y1(
	sIPAddr:= sIpAddr, 
	nTCPPort:= INT_TO_UINT(nTCPPort), 
	nUnitID:= INT_TO_BYTE(nUnitID), 
	mBusAdr:= 4, 
	bEnable:= F_TRIG_Steg8.Q, 
	tTimeout:= tTimeout, 
	bBool:= bVavOutputY1override, 
	bError=> , 
	bBusy=> , 
	bSuccess=> );
	
F_TRIG_Steg9(CLK:= fbReadWriteCoilRegBool_Y1.bBusy, Q=> );
	
	fbReadWriteHoldingRegReal_Y1(
	sIPAddr:= sIpAddr, 
	nTCPPort:= INT_TO_UINT(nTCPPort), 
	nUnitID:= INT_TO_BYTE(nUnitID), 
	mBusAdr:= 6, 
	bEnable:= F_TRIG_Steg9.Q, 
	tTimeout:= tTimeout, 
	rReal:= LIMIT(0,rVavOutputY1override,100), 
	uiFaktor:= 10, 
	bError=> , 
	bBusy=> , 
	bSuccess=> );
	
	F_TRIG_Steg10(CLK:= fbReadWriteHoldingRegReal_Y1.bBusy, Q=> );
		
	//Hantering justeringsvärden
	IF SP4 < -3 THEN
		SP4 := -3;
	END_IF
	
	IF SP4 > 3 THEN
		SP4 := 3;
	END_IF
	
	wWordToWrite := fRealToWord(SP4,10);
			
	fbReadWriteHoldingRegReal_Setpoint(
	sIPAddr:= sIpAddr, 
	nTCPPort:= INT_TO_UINT(nTCPPort), 
	nUnitID:= INT_TO_BYTE(nUnitID), 
	mBusAdr:= 9, 
	bEnable:= F_TRIG_Steg10.Q, 
	tTimeout:= tTimeout, 
	rReal:= wWordToWrite, 
	uiFaktor:= 1, 
	bError=> , 
	bBusy=> , 
	bSuccess=> );
		
//Communication error
	fbKommTof(IN:=FB_MBReadRegs_InputRegs1.bError OR fbReadWriteHoldingRegReal_Sp.bError OR fbReadWriteHoldingRegReal_Offset.bError OR
	fbReadWriteCoilRegBool_Night.bError OR fbReadWriteCoilRegBool_A1.bError OR fbReadWriteHoldingRegReal_A1.bError OR
	fbReadWriteCoilRegBool_A2.bError OR fbReadWriteHoldingRegReal_A2.bError OR
	fbReadWriteCoilRegBool_Y1.bError OR fbReadWriteHoldingRegReal_Y1.bError OR fbReadWriteHoldingRegReal_Setpoint.bError, PT:=T#20S , Q=> , ET=> );
	fbKommTon(bInput:=fbKommTof.Q , tAlarmDelay:=T#20M , bAutoReset:= , bAlarmOutput=> );
	FAULT :=fbKommTon.bAlarmOutput;
		
//Write busy	
	
	bBusy := FB_MBReadRegs_InputRegs1.bBusy OR fbReadWriteHoldingRegReal_Sp.bBusy OR fbReadWriteHoldingRegReal_Offset.bBusy OR
	fbReadWriteCoilRegBool_Night.bBusy OR fbReadWriteCoilRegBool_A1.bBusy OR fbReadWriteHoldingRegReal_A1.bBusy OR
	fbReadWriteCoilRegBool_A2.bBusy OR fbReadWriteHoldingRegReal_A2.bBusy OR
	fbReadWriteCoilRegBool_Y1.bBusy OR fbReadWriteHoldingRegReal_Y1.bBusy OR fbReadWriteHoldingRegReal_Setpoint.bBusy;
	
	oaksgvl.aBModbusBusyFlagga[iModbusLoop,nUnitID] := bBusy;

END_FUNCTION_BLOCK

// oaksModbusLibrary/Produal/Regulatorer/HLS44/fbProdualHLS44_IO
FUNCTION_BLOCK fbProdualHLS44_IO
VAR_INPUT
   rOutput : REAL := 0; //Ingång
END_VAR

VAR_OUTPUT
	{attribute 'OPC.UA.DA' := '1'}
	OP AT %M* : REAL;//Utsignal~wp:[unit]%[format]0
	{attribute 'OPC.UA.DA' := '1'}
	AL8 AT %M* : BOOL;//Utsignal handställd~wp:[alarmoptions]p:3
END_VAR

VAR
	fbAlarm2: fbAlarm;
END_VAR

VAR_INPUT PERSISTENT
	{attribute 'OPC.UA.DA' := '1'}
	M AT %M*: BOOL;//Handställning~wp:
	{attribute 'OPC.UA.DA' := '1'}
	OPM AT %M* : REAL;//Värde handställning~wp:[unit]%[format]0
END_VAR

OP := rOutput;

//Handställningslarm
fbAlarm2(bInput:=M , tAlarmDelay:= , bAutoReset:=TRUE , bAlarmOutput=>AL8 );
	
IF OPM < 0 THEN
	OPM := 0;
END_IF

IF OPM > 100 THEN
	OPM := 100;
END_IF

END_FUNCTION_BLOCK

// oaksModbusLibrary/Produal/Regulatorer/fbProdualHdhmCo2Override
//OAKS AB
//2020-10-12
//Funktionsblock för Produal HDH-M. Inbyggda taggar temp/CO2. Överstyrningsmöjlighet på ugångar Y1-Y4.
//bYxEnable för respektive utgång sätts till TRUE, börvärde sätts 0-100&% till bYxSetpoint.
FUNCTION_BLOCK fbProdualHdhmCo2Override
VAR_INPUT
	sIPAddr : STRING := '127.0.0.1'; 
	nTCPPort : UINT := 502;
	nUnitID : UINT :=1;
	iModbusLoop : INT :=1; //Modbusslinga
	bY1Enable : BOOL := FALSE; //Aktivera skrivning till Y1
	rY1Setpoint AT %M* : REAL := 0; //Börvärde utsignal Y1 (0-100%)
	bY2Enable : BOOL := FALSE; //Aktivera skrivning till Y1
	rY2Setpoint AT %M* : REAL := 0; //Börvärde utsignal Y2 (0-100%)
	bY3Enable : BOOL := FALSE; //Aktivera skrivning till Y1
	rY3Setpoint AT %M* : REAL := 0; //Börvärde utsignal Y3 (0-100%)
	bY4Enable : BOOL := FALSE; //Aktivera skrivning till Y1
	rY4Setpoint AT %M* : REAL := 0; //Börvärde utsignal Y4 (0-100%)
			
END_VAR
VAR_OUTPUT
	PV AT %M*: REAL; //Temperatur~wp:[unit]°C[format]0.0[trendoptions]i:300
	PV1 AT %M* : REAL; //Koldioxidhalt~wp:[unit]ppm[format]0[trendoptions]i:300
	rY1 AT %M* : REAL; //Utsignal Y1 (0-100%)
	rY2 AT %M* : REAL; //Utsignal Y2 (0-100%)
	rY3 AT %M* : REAL; //Utsignal Y3 (0-100%)
	rY4 AT %M* : REAL; //Utsignal Y4 (0-100%)
	PV8 AT %M* : STRING;//Modbus konfiguering~wp:
	FAULT AT %M* : BOOL;//Kommunikationsfel~wp:
	
END_VAR
VAR
	wTemp : WORD;
	bSekvensFlagga : BOOL;
	
	//Coils
	FB_MBReadCoils_Y1: FB_MBReadCoils;
	FB_MBWriteCoils_Y1 : FB_MBWriteCoils;
	bY1EnableRead : BOOL := FALSE;
	
	FB_MBReadCoils_Y2: FB_MBReadCoils;
	FB_MBWriteCoils_Y2 : FB_MBWriteCoils;
	bY2EnableRead : BOOL := FALSE;
	
	FB_MBReadCoils_Y3: FB_MBReadCoils;
	FB_MBWriteCoils_Y3 : FB_MBWriteCoils;	
	bY3EnableRead : BOOL := FALSE;
	
	FB_MBReadCoils_Y4: FB_MBReadCoils;
	FB_MBWriteCoils_Y4 : FB_MBWriteCoils;
	bY4EnableRead : BOOL := FALSE;
	
	//Input registers			
	FB_MBReadRegs_InputRegs1: FB_MBReadInputRegs;
	ArrInputRegs1 : ARRAY [1..7] OF WORD; //Input Regs
	
	//Holding registers
	fbReadWriteHoldingReg_Y1: fbReadWriteHoldingReg;
	fbReadWriteHoldingReg_Y2: fbReadWriteHoldingReg;
	fbReadWriteHoldingReg_Y3: fbReadWriteHoldingReg;
	fbReadWriteHoldingReg_Y4: fbReadWriteHoldingReg;
		
	//Kommunikationsfel
	fbKommTof : tof;
	fbAlarm_1: OaksLibrary.fbAlarm; 
		
	sIP: STRING(255);
	sPort: STRING(255);
	sModbusID: STRING(255);
	sModbusLoop: STRING(255);
	sTemp : STRING(255);
		

END_VAR

//General
	//Offset -1 från modbus-lista.
//Sekvens	
	bSekvensFlagga := oaksGVL.aBModbusSekvens[iModbusLoop] = UINT_TO_INT(nUnitID);
//Modbus konfiguering
	sIP := CONCAT (SIPAddr, '');
	sPort := CONCAT ('<br>Port: ', UINT_TO_STRING(nTCPPort)); 								
	sModbusID := CONCAT('<br>ID: ', UINT_TO_STRING(nUnitID));
	sModbusLoop := CONCAT('<br>Loop: ', INT_TO_STRING(iModbusLoop));	

	sTemp := sIP;
	sTemp := CONCAT(sTemp, sPort);
	sTemp := CONCAT(sTemp, sModbusID);
	sTemp := CONCAT(sTemp, sModbusLoop);
	
	PV8 := sTemp;

///////////////		
//Läs
///////////////		
	
	//Läs Input 1-7
	FB_MBReadRegs_InputRegs1(
	sIPAddr:= sIpAddr, 
	nTCPPort:= INT_TO_UINT(nTCPPort), 
	nUnitID:= INT_TO_BYTE(nUnitID), 
	nQuantity:= 7, 
	nMBAddr:= 0, 
	cbLength:= SIZEOF(ArrInputRegs1), 
	pDestAddr:= ADR(ArrInputRegs1), 
	bExecute:= bSekvensFlagga, 
	tTimeout:= T#3S, 
	bBusy=> , 
	bError=> , 
	nErrId=> , 
	cbRead=> );
	
		//Värden
		PV1 := WORD_TO_REAL(ArrInputRegs1[1]); //1 CO2
		PV := WORD_TO_REAL(ArrInputRegs1[2]) / 10; //2 Temperatur
		//ArrInputRegs1[3]; //3 Fukt
		rY1 := WORD_TO_REAL(ArrInputRegs1[4]) / 10; //4 Utsignal Y1
		rY2 := WORD_TO_REAL(ArrInputRegs1[5]) / 10; //5 Utsignal Y2
		rY3 := WORD_TO_REAL(ArrInputRegs1[6]) / 10; //6 Utsignal Y3
		rY4 := WORD_TO_REAL(ArrInputRegs1[7]) / 10; //7 Utsignal Y4
		
///////////////		
//Skriv
///////////////			

//Läs/Skriv Coils
	
